(* PLC project Automating ships steam boiler, TK TC6_v0200_Example2 v2.0, author Toni Kucic *)
(* stored: creationDateTime 2019-09-29T20:50:27.2524554, version 4.1, modificationDateTime 2019-09-29T20:50:02.7007048, organization TkAutomation *)
(* Visit: https://github.com/tkucic/AutoSteamBoiler for more information. *)

TYPE BistableControlAPI_In_Typ : STRUCT
  DeactivateCmd : BOOL;  (* Deactivate cmd *)
  ActivateCmd : BOOL;  (* Activate cmd *)
END_STRUCT;
END_TYPE

TYPE BistableControlAPI_Out_Typ : STRUCT
  Deactivated : BOOL;  (* Device is deactivated *)
  Activated : BOOL;  (* Device is activated *)
  PositionError : BOOL;  (* TRUE: Object has position error *)
  Status : ARRAY[1..20] OF DINT;  (* 1:Open/Closed/InTransit, 2:OpenFail, 3:CloseFail, 4:FBError, 5:Control Position, 6:OpenCmd, 7:CloseCmd *)
  Icon : STRING;
END_STRUCT;
END_TYPE

TYPE BistableControlHMI_In_Typ : STRUCT
  DeactivateCmd : BOOL;  (* Deactivate cmd *)
  ActivateCmd : BOOL;  (* Activate cmd *)
  SetToAuto : BOOL;  (* Sets control to logic mode *)
  SetToMan : BOOL;  (* Sets control to HMI mode *)
END_STRUCT;
END_TYPE

TYPE BistableControlInit_Typ : STRUCT
  OpenFailDelay : TIME := TIME#6s0ms;  (* Open fail delay *)
  CloseFailDelay : TIME := TIME#6s0ms;  (* Close fail delay *)
  PositionErrorDelay : TIME := TIME#10s0ms;  (* Position error delay *)
  FBs : DWORD := 16#3;  (* B0 - Opened signal in use, B1 - Closed signal in use *)
END_STRUCT;
END_TYPE

TYPE BistableControlIO_In_Typ : STRUCT
  Deactivated : BOOL;  (* IO Open signal feedback from the device *)
  Activated : BOOL;  (* IO Close signal feedback from the device *)
  Tripped : BOOL;
  ReadyToOperate : BOOL := TRUE;
  Remote : BOOL := TRUE;
END_STRUCT;
END_TYPE

TYPE BistableControlIO_Out_Typ : STRUCT
  DeactivateCmd : BOOL;  (* IO deactivate command signal *)
  ActivateCmd : BOOL;  (* IO activate command signal *)
END_STRUCT;
END_TYPE

TYPE BistableIndAPI_Typ : STRUCT
  Deactivated : BOOL;  (* Device is deactivated *)
  Activated : BOOL;  (* Device is activated *)
  PositionError : BOOL;  (* TRUE: Object has position error *)
  Icon : STRING;
END_STRUCT;
END_TYPE

TYPE BistableIndInit_Typ : STRUCT
  PositionErrorDelay : TIME := TIME#10s0ms;  (* Position error alarm delay *)
  FBs : DWORD := 3;  (* B0 - Opened signal in use, B1 - Closed signal in use *)
END_STRUCT;
END_TYPE

TYPE BistableIndIO_In_Typ : STRUCT
  Deactivated : BOOL;  (* Device is deactivated input *)
  Activated : BOOL;  (* Device is activated input *)
  Tripped : BOOL;
END_STRUCT;
END_TYPE

TYPE DutyStandbyClassAPI_IN_Typ : STRUCT

END_STRUCT;
END_TYPE

TYPE DutyStandbyClassAPI_OUT_Typ : STRUCT

END_STRUCT;
END_TYPE

TYPE DutyStandbyClassInit_Typ : STRUCT

END_STRUCT;
END_TYPE

TYPE DutyStandbyClassIO_IN_Typ : STRUCT
  Pump1 : BistableControlIO_In_Typ;
  Pump2 : BistableControlIO_In_Typ;
END_STRUCT;
END_TYPE

TYPE DutyStandbyClassIO_OUT_Typ : STRUCT
  Pump1 : BistableControlIO_Out_Typ;
  Pump2 : BistableControlIO_Out_Typ;
END_STRUCT;
END_TYPE

TYPE TankControlClassAPI_IN_Typ : STRUCT
  LevelRef_pc : REAL;
END_STRUCT;
END_TYPE

TYPE TankControlClassAPI_OUT_Typ : STRUCT
  TankLevel_pc : REAL;
END_STRUCT;
END_TYPE

TYPE TankControlClassInit_Typ : STRUCT
  DrainValve : BistableControlInit_Typ;
  FillingValve : BistableControlInit_Typ;
END_STRUCT;
END_TYPE

TYPE TankControlClassIO_IN_Typ : STRUCT
  DrainValve : BistableControlIO_In_Typ;
  FillingValve : BistableControlIO_In_Typ;
  HLimitSwitch : BOOL;
  LLimitSwitch : BOOL;
  Level_cbm : REAL;
END_STRUCT;
END_TYPE

TYPE TankControlClassIO_OUT_Typ : STRUCT
  DrainValve : BistableControlIO_Out_Typ;
  FillingValve : BistableControlIO_Out_Typ;
END_STRUCT;
END_TYPE

TYPE AI_CFG_Typ : STRUCT
  sigMin : REAL;  (* Minimum value of the signal for scaling integer to real *)
  sigMax : REAL;  (* Maximum value of the signal for scaling integer to real *)
  Scale : REAL;  (* Scaling value of the signal for scaling integer to real *)
END_STRUCT;
END_TYPE

TYPE AI_IO_Typ : STRUCT
  PV_IN : REAL;  (* Input variable *)
  Status : DWORD;  (* Signal status *)
  AlarmHigh : BOOL;  (* High alarm flag *)
  AlarmHighHigh : BOOL;  (* High High alarm flag *)
  AlarmLow : BOOL;  (* Low alarm flag *)
  AlarmLowLow : BOOL;  (* Low Low alarm flag *)
  PV : REAL;  (* Proces variable *)
END_STRUCT;
END_TYPE

TYPE AO_CFG_Typ : STRUCT
  sigMin : REAL;  (* Minimum value of the signal for scaling integer to real *)
  sigMax : REAL;  (* Maximum value of the signal for scaling integer to real *)
  Scale : REAL;  (* Scaling value of the signal for scaling integer to real *)
END_STRUCT;
END_TYPE

TYPE AO_IO_Typ : STRUCT
  PV_IN : REAL;  (* Input variable *)
  Status : DWORD;  (* Signal status *)
  PV : REAL;  (* Proces variable *)
END_STRUCT;
END_TYPE

TYPE DI_CFG_Typ : STRUCT
  dummy1 : BOOL;
  dummy2 : BOOL;
  dummy3 : BOOL;
END_STRUCT;
END_TYPE

TYPE DI_IO_Typ : STRUCT
  Status : DWORD;  (* Signal status *)
  AlarmHigh : BOOL;  (* High alarm flag *)
  AlarmHighHigh : BOOL;  (* High High alarm flag *)
  AlarmLow : BOOL;  (* Low alarm flag *)
  AlarmLowLow : BOOL;  (* Low Low alarm flag *)
  PV : BOOL;  (* Proces variable *)
END_STRUCT;
END_TYPE

TYPE DO_CFG_Typ : STRUCT
  dummy1 : BOOL;
  dummy2 : BOOL;
  dummy3 : BOOL;
END_STRUCT;
END_TYPE

TYPE DO_IO_Typ : STRUCT
  Status : DWORD;  (* Signal status *)
  PV : BOOL;  (* Proces variable *)
END_STRUCT;
END_TYPE

TYPE IO_Typ : STRUCT
  AIS : AIS_Typ;  (* Analog input structure *)
  AOS : AOS_Typ;  (* Analog output structure *)
  DIS : DIS_Typ;  (* Digital input structure *)
  DOS : DOS_Typ;  (* Digital output structure *)
END_STRUCT;
END_TYPE

TYPE LIO : STRUCT
  IgnitionSeq : INT;
  ResetRequired : BOOL;
  FlameEstablished : BOOL;
  SteamCondensation : REAL;
  MasterFWPP : DINT;
  SteamDump : REAL;
  SteamConsumers : REAL;
END_STRUCT;
END_TYPE

TYPE AIS_Typ : STRUCT
  x150_BOILER_WATER_LEVEL : AI_IO_Typ;  (* Boiler water level *)
  x200_FRESH_WATER_STORAGE_TANK_LEVEL : AI_IO_Typ;  (* Fresh water storage tank level *)
  x200_FRESH_WATER_SERVICE_TANK_LEVEL : AI_IO_Typ;  (* Fresh water service tank level *)
  x300_HFO_HEATING_SYSTEM_CONSUMPTION : AI_IO_Typ;  (* HFO Heating system consumption *)
  x300_HVAC_SYSTEM_CONSUMPTION : AI_IO_Typ;  (* HVAC system consumption *)
  x300_OPERATIONAL_CONSUMERS_CONSUMPTION : AI_IO_Typ;  (* Operational consumers consumption *)
  x300_SYSTEM_STEAM_PRESSURE : AI_IO_Typ;  (* System steam pressure *)
END_STRUCT;
END_TYPE

TYPE AOS_Typ : STRUCT
  x150_BOILER_WATER_FEED_REGULATION_VALVE_SETPOINT : AO_IO_Typ;  (* Boiler water feed regulation valve setpoint *)
  x150_STEAM_DUMP_VALVE_SETPOINT : AO_IO_Typ;  (* Steam dump valve setpoint *)
  x100_AIR_VALVE_SETPOINT : AO_IO_Typ;  (* Air valve setpoint *)
  x100_FUEL_VALVE_SETPOINT : AO_IO_Typ;  (* Fuel valve setpoint *)
END_STRUCT;
END_TYPE

TYPE DOS_Typ : STRUCT
  x200_FW_SERVICE_PUMP1_STARTCMD : DO_IO_Typ;  (* Fresh water service pump 1 start command *)
  x200_FW_SERVICE_PUMP1_STOPCMD : DO_IO_Typ;  (* Fresh water service pump 1 stop command *)
  x200_FW_SERVICE_PUMP2_STARTCMD : DO_IO_Typ;  (* Fresh water service pump 2 start command *)
  x200_FW_SERVICE_PUMP2_STOPCMD : DO_IO_Typ;  (* Fresh water service pump 2 stop command *)
  x200_FW_STORAGE_TANK_DRAINVALVE_CLOSECMD : DO_IO_Typ;  (* Fresh water storage tank drain valve close command *)
  x200_FW_STORAGE_TANK_DRAINVALVE_OPENCMD : DO_IO_Typ;  (* Fresh water storage tank drain valve open command *)
  x200_FW_STORAGE_TANK_FILLVALVE_CLOSECMD : DO_IO_Typ;  (* Fresh water storage tank filling valve close command *)
  x200_FW_STORAGE_TANK_FILLVALVE_OPENCMD : DO_IO_Typ;  (* Fresh water storage tank filling valve open command *)
  x200_FW_SERVICE_TANK_DRAINVALVE_CLOSECMD : DO_IO_Typ;  (* Fresh water service tank drain valve close command *)
  x200_FW_SERVICE_TANK_DRAINVALVE_OPENCMD : DO_IO_Typ;  (* Fresh water service tank drain valve open command *)
  x200_FW_SERVICE_TANK_FILLVALVE_CLOSECMD : DO_IO_Typ;  (* Fresh water service tank filling valve close command *)
  x200_FW_SERVICE_TANK_FILLVALVE_OPENCMD : DO_IO_Typ;  (* Fresh water service tank filling valve open command *)
  x100_IGNITOR_ACTIVATE_CMD : DO_IO_Typ;  (* Ignitor activate cmd *)
  x100_BLOWER_MOTOR_START_CMD : DO_IO_Typ;  (* Blower motor start cmd *)
  x100_MAIN_FUEL_VALVE_CLOSE_CMD : DO_IO_Typ;  (* Main fuel valve close cmd *)
  x100_MAIN_FUEL_VALVE_OPEN_CMD : DO_IO_Typ;  (* Main fuel valve open cmd *)
  x300_HFO_HEATING_VALVE_CLOSE_CMD : DO_IO_Typ;  (* HFO heating valve close cmd *)
  x300_HFO_HEATING_VALVE_OPEN_CMD : DO_IO_Typ;  (* HFO heating valve open cmd *)
  x300_HVAC_HEATING_VALVE_CLOSE_CMD : DO_IO_Typ;  (* HVAC heating valve close cmd *)
  x300_HVAC_HEATING_VALVE_OPEN_CMD : DO_IO_Typ;  (* HVAC heating valve open cmd *)
  x300_OPERATIONAL_CONSUMERS_VALVE_CLOSE_CMD : DO_IO_Typ;  (* Operational consumers valve close cmd *)
  x300_OPERATIONAL_CONSUMERS_VALVE_OPEN_CMD : DO_IO_Typ;  (* Operational consumers valve open cmd *)
END_STRUCT;
END_TYPE

TYPE DIS_Typ : STRUCT
  x100_PHOTOCELL1_ACTIVE : DI_IO_Typ;  (* Photocell1Active *)
  x100_PHOTOCELL2_ACTIVE : DI_IO_Typ;  (* Photocell2Active *)
  x100_BURNER_DOOR_OPEN : DI_IO_Typ;  (* Burner door open *)
  x100_IGNITION_COIL_ACTIVATED : DI_IO_Typ;  (* Ignition coil activated *)
  x100_MAIN_FUEL_VALVE_CLOSED : DI_IO_Typ;  (* Main fuel valve closed *)
  x100_MAIN_FUEL_VALVE_OPEN : DI_IO_Typ;  (* Main fuel valve open *)
  x200_FW_STORAGE_TK_HLIMITSWITCH : DI_IO_Typ;  (* Fresh water storage tank high limit switch active *)
  x200_FW_STORAGE_TK_LLIMITSWITCH : DI_IO_Typ;  (* Fresh water storage tank low limit switch active *)
  x200_FW_SERVICE_PUMP2_RUNNING : DI_IO_Typ;  (* Fresh water service pump 2 running *)
  x200_FW_SERVICE_PUMP2_STOPPED : DI_IO_Typ;  (* Fresh water service pump 2 stopped *)
  x200_FW_SERVICE_PUMP2_READY : DI_IO_Typ;  (* Fresh water service pump 2 ready *)
  x200_FW_SERVICE_PUMP2_TRIPPED : DI_IO_Typ;  (* Fresh water service pump 2 tripped *)
  x200_FW_SERVICE_PUMP2_REMOTE : DI_IO_Typ;  (* Fresh water service pump 2 remote *)
  x200_FW_SERVICE_PUMP1_RUNNING : DI_IO_Typ;  (* Fresh water service pump 1 running *)
  x200_FW_SERVICE_PUMP1_STOPPED : DI_IO_Typ;  (* Fresh water service pump 1 stopped *)
  x200_FW_SERVICE_PUMP1_READY : DI_IO_Typ;  (* Fresh water service pump 1 ready *)
  x200_FW_SERVICE_PUMP1_TRIPPED : DI_IO_Typ;  (* Fresh water service pump 1 tripped *)
  x200_FW_SERVICE_PUMP1_REMOTE : DI_IO_Typ;  (* Fresh water service pump 1 remote *)
  x200_FW_STORAGE_TK_DRAINVALVE_CLOSED : DI_IO_Typ;  (* Fresh water storage tank drain valve closed *)
  x200_FW_STORAGE_TK_DRAINVALVE_OPENED : DI_IO_Typ;  (* Fresh water storage tank drain valve opened *)
  x200_FW_STORAGE_TK_DRAINVALVE_READY : DI_IO_Typ;  (* Fresh water storage tank drain valve ready *)
  x200_FW_STORAGE_TK_DRAINVALVE_REMOTE : DI_IO_Typ;  (* Fresh water storage tank drain valve remote *)
  x200_FW_STORAGE_TK_FILLVALVE_CLOSED : DI_IO_Typ;  (* Fresh water storage tank filling valve closed *)
  x200_FW_STORAGE_TK_FILLVALVE_OPENED : DI_IO_Typ;  (* Fresh water storage tank filling valve opened *)
  x200_FW_STORAGE_TK_FILLVALVE_READY : DI_IO_Typ;  (* Fresh water storage tank filling valve ready *)
  x200_FW_STORAGE_TK_FILLVALVE_REMOTE : DI_IO_Typ;  (* Fresh water storage tank filling valve remote *)
  x200_FW_SERVICE_TK_HLIMITSWITCH : DI_IO_Typ;  (* Fresh water service tank high limit switch active *)
  x200_FW_SERVICE_TK_LLIMITSWITCH : DI_IO_Typ;  (* Fresh water service tank low limit switch active *)
  x200_FW_SERVICE_TK_DRAINVALVE_CLOSED : DI_IO_Typ;  (* Fresh water service tank drain valve closed *)
  x200_FW_SERVICE_TK_DRAINVALVE_OPENED : DI_IO_Typ;  (* Fresh water service tank drain valve opened *)
  x200_FW_SERVICE_TK_DRAINVALVE_READY : DI_IO_Typ;  (* Fresh water service tank drain valve ready *)
  x200_FW_SERVICE_TK_DRAINVALVE_REMOTE : DI_IO_Typ;  (* Fresh water service tank drain valve remote *)
  x200_FW_SERVICE_TK_FILLVALVE_CLOSED : DI_IO_Typ;  (* Fresh water service tank filling valve closed *)
  x200_FW_SERVICE_TK_FILLVALVE_OPENED : DI_IO_Typ;  (* Fresh water service tank filling valve opened *)
  x200_FW_SERVICE_TK_FILLVALVE_READY : DI_IO_Typ;  (* Fresh water service tank filling valve ready *)
  x200_FW_SERVICE_TK_FILLVALVE_REMOTE : DI_IO_Typ;  (* Fresh water service tank filling valve remote *)
  x300_OPERATIONAL_CONSUMERS_VALVE_OPEN : DI_IO_Typ;  (* Operational consumers valve open *)
  x300_HFO_HEATING_VALVE_CLOSED : DI_IO_Typ;  (* HFO heating valve closed *)
  x300_HFO_HEATING_VALVE_OPEN : DI_IO_Typ;  (* HFO heating valve open *)
  x300_HVAC_HEATING_VALVE_CLOSED : DI_IO_Typ;  (* HVAC heating valve closed *)
  x300_HVAC_HEATING_VALVE_OPEN : DI_IO_Typ;  (* HVAC heating valve open *)
  x300_OPERATIONAL_CONSUMERS_VALVE_CLOSED : DI_IO_Typ;  (* Operational consumers valve closed *)
  x900_EMERGENCY_STOP : DI_IO_Typ;  (* Emergency stop *)
  x900_SYSTEM_REMOTE_SWITCH : DI_IO_Typ;  (* SystemRemote switch *)
END_STRUCT;
END_TYPE

TYPE SimCFG : STRUCT
  BlinkFreq : TIME := TIME#500ms;
  FWTankLSHighTrig : REAL := 85;
  FWTankLSHighHighTrig : REAL := 95;
  FWTankLSLowTrig : REAL := 15;
  FWTankLSLowLowTrig : REAL := 5;
  SteamFactor : REAL := 0.021;
  ReliefValveOpeningSP : REAL := 35;
  Inflow : REAL := 0.11;
  WaterEvapFactor : REAL := 0.06;
  MaxDump : REAL := 1;
  OverpressureMultiplier : REAL := 1;
  DrainTankMultiplier : REAL := 0.5;
  PCell1DetectDelay : TIME := TIME#500ms;
  PCell2DetectDelay : TIME := TIME#1s0ms;
  ValveOperatingTime : TIME := TIME#3s0ms;
  LostWaterOnConsumers : REAL := 0.1;
END_STRUCT;
END_TYPE

TYPE CFG_Typ : STRUCT
  FWTankHighLimit : REAL := 90;  (* High water level limit *)
  FWTankLowLimit : REAL := 30;  (* Low water level limit *)
  FWTankLowTrip : REAL := 15;
  FWTankLowAlarmDelay : TIME := TIME#1s0ms;
  SteamPressureSP : REAL := 7;  (* Setpoint for system steam pressure *)
  FWServiceTKSP : REAL := 70;  (* Setpoint for the FW Service tank water level *)
  SteamPressHighTrip : REAL := 45;
  SteamPressHighLimit : REAL := 8.5;  (* High steam pressure limit *)
  SteamPressLowLimit : REAL := 1;  (* Low steam pressure limit *)
  SteamPressHighAlarmDelay : TIME := TIME#1s0ms;
  FuelValveStart_pc : REAL := 10;  (* Starting valve opening upon ignition sequence *)
  DualPumpsTimer : TIME := TIME#5s0ms;  (* Time for FW pumps to run in paralel during sw/o *)
  BlowingOutTime : TIME := TIME#10s0ms;  (* Time for safety blow out of burner *)
  IgnitionFailDelay : TIME := TIME#5s0ms;  (* Time before ignition fail occurs *)
  MainFuelValveOperationDelay : TIME := TIME#5s0ms;
  F_PID_P : REAL := 1.5;
  F_PID_I : REAL := 0.9;
  F_PID_D : REAL := 0;
  F_PID_Offset : REAL := 0;
  F_PID_OutMIN : REAL := 2.1;
  F_PID_OutMAX : REAL := 100;
  AirToFuelRatio : REAL := 1.25;
  W_PID_P : REAL := 1.5;
  W_PID_I : REAL := 0.9;
  W_PID_D : REAL := 0;
  W_PID_Offset : REAL := 0;
  HFOConsumerNominal : REAL := 1;
  HFOHeatValveOperDelay : TIME := TIME#5s0ms;
  HVACConsumerNominal : REAL := 0.5;
  HVACHeatValveOperDelay : TIME := TIME#5s0ms;
  OperConsumerNominal : REAL := 0.65;
  OperConsValveOperDelay : TIME := TIME#5s0ms;
  S_PID_P : REAL := -1.5;
  S_PID_I : REAL := 0.9;
  S_PID_D : REAL := 0;
  TxtRemote : STRING := 'REMOTE';
  TxtManual : STRING := 'MANUAL';
  TxtOvrFl : STRING := 'FW Tank overflowing';
  TxtFWTkEmpty : STRING := 'FW Tank empty';
  TxtSysReady : STRING := 'System ready for operation';
  TxtSysBlow : STRING := 'System blowout begun';
  TxtIgnite : STRING := 'Igniting burner';
  TxtSysRun : STRING := 'System running';
  TxtIgnFail : STRING := 'Ignition failed';
  TxtEmcyStp : STRING := 'Emergency stop active';
  TxtAbort : STRING := 'Operation aborted by user';
  TxtSysNotReady : STRING := 'System not ready';
END_STRUCT;
END_TYPE

TYPE Vars : STRUCT
  CFG : CFG_Typ;
  dummy1 : BOOL;
  dummy2 : BOOL;
END_STRUCT;
END_TYPE

FUNCTION_BLOCK BurnerControlClass

            
          
END_FUNCTION_BLOCK

FUNCTION_BLOCK fbAuxDevCtrl
  VAR
    ChangeOverTrig : R_TRIG;
    DualPumpsTimer : TOn;
    WaterLevelCTRL : PID;
    vManual : REAL;
    vPIDOFF : BOOL;
    vReset : BOOL;
    vLimitsActive : BOOL;
    vPIDOverflow : BOOL;
  END_VAR
  VAR RETAIN
    vMasterFWPP : INT := 1;
    vAutoStopFWPump2 : BOOL;
    vAutoStartFWPump2 : BOOL;
    vAutoStopFWPump1 : BOOL;
    vAutoStartFWPump1 : BOOL;
    vFWTkSP : REAL := 75;
  END_VAR

            // (* Switch Water level PID off if tank is overflowing *)
// vPIDOFF := GVL.IO.DIS.FWTankLSHighHigh OR GVL.IO.AIS.FWTank_Level > GVL.CFG_Typ.FWTankHighLimit;
// 
// (* Change over functionality. This switches the pumps.*)
// ChangeOverTrig(CLK:=GVL.IO.DIS.FWChangeOverPP);
// 
// IF vMasterFWPP = 1 AND ChangeOverTrig.Q THEN
// 	vMasterFWPP := 2;
// ELSIF vMasterFWPP = 2 AND ChangeOverTrig.Q THEN
// 	vMasterFWPP := 1;
// END_IF;
// 
// (* Automatic regulation of fresh water service tanks level *)
// IF GVL.IO.DIS.RemoteFWPP THEN
// 	vAutoStopFWPump1 := (vMasterFWPP = 1) AND (GVL.IO.DIS.FWTankLSHigh OR GVL.IO.DIS.FWTankLSHighHigh) AND GVL.IO.DOS_Typ.FWPump1;
// 	vAutoStartFWPump1 := (vMasterFWPP = 1) AND (GVL.IO.DIS.FWTankLSLow OR GVL.IO.DIS.FWTankLSLowLow) AND NOT GVL.IO.DOS_Typ.FWPump1;
// 	vAutoStopFWPump2 := (vMasterFWPP = 2) AND (GVL.IO.DIS.FWTankLSHigh OR GVL.IO.DIS.FWTankLSHighHigh) AND GVL.IO.DOS_Typ.FWPump2;
// 	vAutoStartFWPump2 := (vMasterFWPP = 2) AND (GVL.IO.DIS.FWTankLSLow OR GVL.IO.DIS.FWTankLSLowLow) AND NOT GVL.IO.DOS_Typ.FWPump2;
// ELSE
// 	vAutoStopFWPump1 := (vMasterFWPP = 1) AND (GVL.IO.DIS.FWManStop OR GVL.IO.DIS.FWTankLSHighHigh) AND GVL.IO.DOS_Typ.FWPump1;
// 	vAutoStartFWPump1 := (vMasterFWPP = 1) AND GVL.IO.DIS.FWManStart AND NOT GVL.IO.DOS_Typ.FWPump1;
// 	vAutoStopFWPump2 := (vMasterFWPP = 2) AND (GVL.IO.DIS.FWManStop OR GVL.IO.DIS.FWTankLSHighHigh) AND GVL.IO.DOS_Typ.FWPump2;
// 	vAutoStartFWPump2 := (vMasterFWPP = 2) AND GVL.IO.DIS.FWManStart AND NOT GVL.IO.DOS_Typ.FWPump2;
// END_IF
// 
// (*Pumps run paralel for some time to not lose pressure *)
// IF vMasterFWPP = 2 AND GVL.IO.DIS.FWServicePump1=1 THEN
// 	GVL.IO.DOS_Typ.FWPump2 := TRUE;
// 
// 	DualPumpsTimer(IN:=TRUE, PT:=GVL.CFG_Typ.DualPumpsTimer);
// 	IF DualPumpsTimer.Q THEN
// 		GVL.IO.DOS_Typ.FWPump1 := FALSE;
// 		DualPumpsTimer(IN:=FALSE);
// 	END_IF
// ELSIF vAutoStartFWPump1 THEN
// 	GVL.IO.DOS_Typ.FWPump1 := TRUE;
// ELSIF vAutoStopFWPump1 THEN
// 	GVL.IO.DOS_Typ.FWPump1 := FALSE;
// END_IF
// 
// IF vMasterFWPP = 1 AND GVL.IO.DIS.FWServicePump2=1 THEN
// 	GVL.IO.DOS_Typ.FWPump1 := TRUE;
// 	
// 	DualPumpsTimer(IN:=TRUE, PT:=GVL.CFG_Typ.DualPumpsTimer);
// 	IF DualPumpsTimer.Q THEN
// 		GVL.IO.DOS_Typ.FWPump2 := FALSE;
// 		DualPumpsTimer(IN:=FALSE);
// 	END_IF
// ELSIF vAutoStartFWPump2 THEN
// 	GVL.IO.DOS_Typ.FWPump2 := TRUE;
// ELSIF vAutoStopFWPump2 THEN
// 	GVL.IO.DOS_Typ.FWPump2 := FALSE;
// END_IF
// 
// WaterLevelCTRL(
// 	ACTUAL:= GVL.IO.AIS.FWTank_Level, 
// 	SET_POINT:= GVL.CFG_Typ.FWServiceTKSP, 
// 	KP:= GVL.CFG_Typ.W_PID_P, 
// 	TN:= GVL.CFG_Typ.W_PID_I, 
// 	TV:= GVL.CFG_Typ.W_PID_D, 
// 	Y_MANUAL:= 0, 
// 	Y_OFFSET:= GVL.CFG_Typ.W_PID_Offset, 
// 	Y_MIN:= 0, 
// 	Y_MAX:= 100, 
// 	MANUAL:= vPIDOFF, 
// 	RESET:= vReset, 
// 	Y=> GVL.IO.AOS.FWTkRegValve, 
// 	LIMITS_ACTIVE=> vLimitsActive, 
// 	OVERFLOW=> vPIDOverflow);
// 
// (* Send system status to other programs *)
// GVL.LIO.MasterFWPP := vMasterFWPP;
          
END_FUNCTION_BLOCK

FUNCTION_BLOCK fbBoilerSystem

            
          
END_FUNCTION_BLOCK

FUNCTION_BLOCK fbStateMachine
  VAR
    BlowingTimeTimer : TON;
    DelayTimer : TON;
    AutoStartSR : SR;
    vFlameOut : BOOL;
    vOpenMainFuelValveCmd : BOOL;  (* MainFuelValveCtrl: OnOffValve_Object; *)
    vCloseMainFuelValveCmd : BOOL;
    vCloseMainFuelValveHMI : BOOL;
    vOpenMainFuelValveHMI : BOOL;
    vSetMainFuelValveToAuto : BOOL;
    vSetMainFuelValveToMan : BOOL;
    vMainFuelValveStatus : ARRAY[1..20] OF DINT;
    vMainFuelValveIcon : STRING;
    vMainFuelValveButton : BOOL;
  END_VAR
  VAR CONSTANT
    cStateNotReady : INT := 0;
    cStateStandby : INT := 1;
    cStateAirBlowing : INT := 2;
    cStateIgnition : INT := 3;
    cStateSystemIgnited : INT := 4;
    cStateIgnitionFail : INT := 10;
    cStateEmergencyStop : INT := 11;
    cStateUserAbort : INT := 12;
  END_VAR
  VAR RETAIN
    vSequence : INT := 0;
    vSequenceDone : INT;
    vIgnTimerStart : BOOL;
    vIgnSeqStart : BOOL;
    vMessage : STRING(INT#50);
    vResetRequired : BOOL;
    vAutoStart : BOOL;
    vFWTankLowTrip : BOOL;
    vHighPressureTrip : BOOL;
  END_VAR

            // (*******************************************)
// (* 0 - System not ready                    *)
// (* 1 - System standby                      *)
// (* 2 - Air blowing                         *)
// (* 3 - Ignition                            *)
// (* 4 - System ignited                      *)
// (* 10 - Ignition fail                      *)
// (* 11 - Emergency stop                     *)
// (* 12 - User abort                         *)
// (*******************************************)
// 
// (* Safety tripping *)
// 
// vFWTankLowTrip := GVL.IO.AIS.FWTank_Level < GVL.CFG_Typ.FWTankLowTrip AND (vSequence = cStateSystemIgnited);
// 
// vHighPressureTrip := GVL.IO.AIS.SteamPressure > GVL.CFG_Typ.SteamPressHighLimit;
// 
// vFlameOut := (vSequence = cStateSystemIgnited) AND NOT (GVL.IO.DIS.Photocell1 OR GVL.IO.DIS.Photocell2);
// 
// IF vFWTankLowTrip OR vHighPressureTrip OR vFlameOut OR GVL.IO.DIS.BurnerOpen THEN
// 	vSequence := cStateEmergencyStop;
// END_IF
// 
// IF  NOT GVL.IO.DIS.EmcyStopPB THEN
// 	vSequence := cStateEmergencyStop;
// END_IF
// 
// AutoStartSR(Set1:= (GVL.IO.AIS.SteamPressure < GVL.CFG_Typ.SteamPressureSP AND vSequence = cStateStandby), 
// 			Reset:= vSequence <> cStateStandby,
// 			Q1 => vAutoStart);
// 
// CASE vSequence OF
// 		10,11,12: vResetRequired := TRUE;
// ELSE
// 		vResetRequired := FALSE;
// END_CASE
// 
// CASE vSequence OF
// 	
// 	(* System not ready *)
// 	0: vMessage := GVL.CFG_Typ.TxtSysNotReady;
// 		IF GVL.IO.AIS.FWTank_Level > GVL.CFG_Typ.FWTankLowLimit AND GVL.IO.AIS.SteamPressure < GVL.CFG_Typ.SteamPressHighLimit THEN
// 			vSequence := cStateStandby;
// 		END_IF
// 		vSequenceDone := 0;
// 
// 	(* System standby *)
// 	1:  vMessage := GVL.CFG_Typ.TxtSysReady;
// 		IF vAutoStart AND GVL.IO.DIS.RemoteSW THEN
// 			vSequence := cStateAirBlowing;
// 		ELSIF GVL.IO.DIS.ManStartPB THEN
// 			vSequence := cStateAirBlowing;
// 		END_IF
// 		vSequenceDone := 1;
// 		
// 	(* Air blowing and opening valves *)	
// 	2:  vMessage := GVL.CFG_Typ.TxtSysBlow;		
// 		BlowingTimeTimer(IN:=vSequenceDone = 2, PT := GVL.CFG_Typ.BlowingOutTime);
// 		
// 		vOpenMainFuelValveCmd := NOT GVL.IO.DIS.MainFuelValveOpen AND GVL.IO.DIS.RemoteSW;
// 		vCloseMainFuelValveCmd := FALSE;
// 		
// 		GVL.IO.DOS_Typ.AirBlowerMotor := TRUE;
// 		
// 		IF GVL.IO.DIS.StopPB THEN
// 			vSequence := cStateUserAbort;
// 		END_IF;	
// 		
// 		IF BlowingTimeTimer.Q AND GVL.IO.DIS.MainFuelValveOpen THEN
// 			vSequence := cStateIgnition;
// 		ELSIF BlowingTimeTimer.Q AND NOT GVL.IO.DIS.MainFuelValveOpen THEN
// 			vSequence := cStateIgnitionFail;
// 		END_IF
// 		vSequenceDone := 2;
// 	
// 	(* Ignition *)
// 	3:  vMessage := GVL.CFG_Typ.TxtIgnite;
// 		IF GVL.IO.DIS.StopPB THEN
// 			vSequence := cStateUserAbort;
// 		END_IF;	
// 	    vIgnSeqStart :=  vIgnSeqStart OR (GVL.IO.DIS.RemoteSW) OR (GVL.IO.DIS.ManIgnite);
// 		vIgnTimerStart := vSequenceDone = 3 AND vIgnSeqStart;
// 
// 		DelayTimer(IN := vIgnTimerStart, PT := GVL.CFG_Typ.IgnitionFailDelay);
// 		IF DelayTimer.Q THEN
// 			vSequence := cStateIgnitionFail;
// 		END_IF
// 		IF vIgnSeqStart THEN
// 			GVL.IO.DOS_Typ.Ignitor := TRUE;
// 			IF GVL.IO.DIS.Photocell1 OR GVL.IO.DIS.Photocell2 THEN
// 				vSequence := cStateSystemIgnited;
// 				GVL.IO.DIS.ManIgnite := FALSE;
// 				GVL.IO.DOS_Typ.Ignitor := FALSE;
// 				vIgnSeqStart := FALSE;
// 			END_IF
// 		END_IF;
// 		vSequenceDone := 3;
// 		
// 	(* System ignited *)	
// 	4:	vMessage := GVL.CFG_Typ.TxtSysRun;
// 		IF GVL.IO.DIS.StopPB THEN
// 			vSequence := cStateUserAbort;
// 		END_IF;	
// 		vSequenceDone := 4;
// 		
// 	(* Ignition fail *)	
// 	10: vMessage := GVL.CFG_Typ.TxtIgnFail;
// 		GVL.IO.DOS_Typ.Ignitor := FALSE;		
// 		vOpenMainFuelValveCmd := FALSE;
// 		vCloseMainFuelValveCmd := TRUE;
// 		IF GVL.IO.DIS.Reset THEN
// 			vSequence := cStateNotReady;
// 		END_IF
// 		vSequenceDone := 10;
// 		
// 	(* Emergency stop *)	
// 	11: vMessage := GVL.CFG_Typ.TxtEmcyStp;
// 		GVL.IO.DOS_Typ.Ignitor := FALSE;		
// 		vOpenMainFuelValveCmd := FALSE;
// 		vCloseMainFuelValveCmd := TRUE;
// 		IF GVL.IO.DIS.Reset AND GVL.IO.DIS.EmcyStopPB THEN
// 			vSequence := cStateNotReady;
// 		END_IF	
// 		vSequenceDone := 11;
// 		
// 	(* User abort *)	
// 	12:	vMessage := GVL.CFG_Typ.TxtAbort;
// 		BlowingTimeTimer(IN := vSequenceDone = 12, PT := GVL.CFG_Typ.BlowingOutTime);
// 		IF NOT BlowingTimeTimer.Q THEN
// 			GVL.IO.DOS_Typ.AirBlowerMotor := TRUE;
// 		ELSE
// 			GVL.IO.DOS_Typ.AirBlowerMotor := FALSE;
// 		END_IF
// 		IF GVL.IO.DIS.Reset THEN
// 			vSequence := cStateNotReady;
// 		END_IF
// 		GVL.IO.DOS_Typ.Ignitor := FALSE;	
// 		vOpenMainFuelValveCmd := FALSE;
// 		vCloseMainFuelValveCmd := TRUE;
// 		vSequenceDone := 12;
// ELSE
// 	vSequence := cStateNotReady;
// END_CASE
// 
// IF vSequence <> 3 THEN
// 	GVL.IO.DIS.ManIgnite := FALSE;
// END_IF;
// 
// (* Send system status to other programs *)
// GVL.LIO.IgnitionSeq := vSequence;
// GVL.LIO.ResetRequired := vResetRequired;
// 
// (* Fuel Valve controllers *)
// 
// MainFuelValveCtrl(
// 	iOpenedFB:= GVL.IO.DIS.MainFuelValveOpen, 
// 	iClosedFB:= GVL.IO.DIS.MainFuelValveClosed, 
// 	OpenAutoCmd:= vOpenMainFuelValveCmd, 
// 	CloseAutoCmd:= vCloseMainFuelValveCmd, 
// 	OpenCmdHMI:= vOpenMainFuelValveHMI, 
// 	CloseCmdHMI:= vCloseMainFuelValveHMI, 
// 	SetToAuto:= vSetMainFuelValveToAuto, 
// 	SetToMan:= vSetMainFuelValveToMan, 
// 	cfgOpenFailDelay:= GVL.CFG_Typ.MainFuelValveOperationDelay, 
// 	cfgCloseFailDelay:= GVL.CFG_Typ.MainFuelValveOperationDelay, 
// 	cfgFBErrorDelay:= GVL.CFG_Typ.MainFuelValveOperationDelay, 
// 	ValveStatus=> vMainFuelValveStatus, 
// 	ValveIcon=> vMainFuelValveIcon, 
// 	qOpenCmd=> GVL.IO.DOS_Typ.FuelValveOpenCmd, 
// 	qCloseCmd=> GVL.IO.DOS_Typ.FuelValveCloseCmd);

          
END_FUNCTION_BLOCK

FUNCTION_BLOCK fbSteamControl
  VAR
    FuelController : PID;
    SteamDumpController : PID;
    rtManUp : R_TRIG;
    rtManDown : R_TRIG;
    vMan_Y : REAL;
    vHFOHeatOpenCmdHMI : BOOL;  (* HFOHeatValve: OnOffValve_Object; HVACHeatValve: OnOffValve_Object; OperConsValve: OnOffValve_Object; *)
    vHFOHeatCloseCmdHMI : BOOL;
    vHFOHeatSetToAuto : BOOL;
    vHFOHeatSetToMan : BOOL;
    vHFOHeatValveStatus : ARRAY[1..20] OF DINT;
    vHFOHeatValveIcon : STRING;
    vHFOHeatValveButton : BOOL;
    vHVACHeatOpenCmdHMI : BOOL;
    vHVACHeatCloseCmdHMI : BOOL;
    vHVACHeatSetToMan : BOOL;
    vHVACHeatValveStatus : ARRAY[1..20] OF DINT;
    vHVACHeatValveIcon : STRING;
    vHVACHeatValveButton : BOOL;
    vOperConsOpenCmdHMI : BOOL;
    vOperConsCloseCmdHMI : BOOL;
    vOperConsSetToMan : BOOL;
    vOperConsValveStatus : ARRAY[1..20] OF DINT;
    vOperConsValveIcon : STRING;
    vOperConsValveButton : BOOL;
    vHFOHeatOpenAutoCmd : BOOL;
    vHFOHeatCloseAutoCmd : BOOL;
    vHVACHeatValveOpenAutoCmd : BOOL;
    vHVACHeatValveCloseAutoCmd : BOOL;
    vHVACHeatSetToAuto : BOOL;
    vOperConsValveOpenAutoCmd : BOOL;
    vOperConsValveCloseAutoCmd : BOOL;
    vOperConsSetToAuto : BOOL;
  END_VAR
  VAR RETAIN
    vPIDManual : BOOL;
    vOverflow : BOOL;
    vPIDLimitActive : BOOL;
  END_VAR

            // IF GVL.LIO.IgnitionSeq > 4 OR GVL.LIO.IgnitionSeq = 0 THEN
// 	(* Switch off fuel valve *)
// 	vPIDManual	:= TRUE;
// 	vMan_Y		:= 0;
// 
// ELSIF GVL.LIO.IgnitionSeq = 3 THEN
// 	(* Stabilize ignition *)
// 	vPIDManual := TRUE;
// 	vMan_Y 	   := GVL.SysCFG.FuelValveStart_pc;
// 
// ELSIF GVL.LIO.IgnitionSeq = 4 THEN
// 	IF GVL.IO.DIS.RemoteSW THEN
// 		vPIDManual := FALSE;
// 		vMan_Y := GVL.IO.AOS.FuelValve;
// 	ELSIF NOT GVL.IO.DIS.RemoteSW THEN
// 		vPIDManual := TRUE;
// 		rtManUp(CLK:=GVL.IO.DIS.ManLoadUP);
// 		rtManDown(CLK:=GVL.IO.DIS.ManLoadDown);
// 	
// 		IF rtManUp.Q THEN
// 			vMan_Y := vMan_Y + 1;
// 		END_IF
// 		IF rtManDown.Q THEN
// 			vMan_Y := vMan_Y - 1;
// 		END_IF
// 	END_IF
// 		
// ELSE
// 	vPIDManual	:= TRUE;
// 	vMan_Y		:= 0;
// END_IF;
// 
// FuelController(
// 	ACTUAL:= GVL.IO.AIS.SteamPressure, 
// 	SET_POINT:= GVL.SysCFG.SteamPressureSP , 
// 	KP:= GVL.SysCFG.F_PID_P, 
// 	TN:= GVL.SysCFG.F_PID_I, 
// 	TV:= GVL.SysCFG.F_PID_D, 
// 	Y_MANUAL:= vMan_Y, 
// 	Y_OFFSET:= GVL.SysCFG.F_PID_Offset, 
// 	Y_MIN:= GVL.SysCFG.F_PID_OutMIN, 
// 	Y_MAX:= GVL.SysCFG.F_PID_OutMAX,
// 	MANUAL := vPIDManual,
// 	RESET:=FALSE , 
// 	Y=> GVL.IO.AOS.FuelValve, 
// 	LIMITS_ACTIVE=> vPIDLimitActive, 
// 	OVERFLOW=>vOverflow );
// 
// SteamDumpController(
// 	ACTUAL:= GVL.IO.AIS.SteamPressure, 
// 	SET_POINT:= GVL.SysCFG.SteamPressureSP , 
// 	KP:= GVL.SysCFG.S_PID_P, 
// 	TN:= GVL.SysCFG.S_PID_I, 
// 	TV:= GVL.SysCFG.S_PID_D, 
// 	Y_MIN:= 0, 
// 	Y_MAX:= 100,
// 	Y=> GVL.IO.AOS.SteamDumpValve);
// 	
// (* Consumer valve handling *)
// HFOHeatValve(
// 	iOpenedFB:= GVL.IO.DIS.HFOHeatValveOpen , 
// 	iClosedFB:= GVL.IO.DIS.HFOHeatValveClosed, 
// 	OpenAutoCmd:= vHFOHeatOpenAutoCmd, 
// 	CloseAutoCmd:= vHFOHeatCloseAutoCmd, 
// 	OpenCmdHMI:= vHFOHeatOpenCmdHMI, 
// 	CloseCmdHMI:= vHFOHeatCloseCmdHMI, 
// 	SetToAuto:= vHFOHeatSetToAuto, 
// 	SetToMan:= vHFOHeatSetToMan, 
// 	cfgOpenFailDelay:= GVL.SysCFG.HFOHeatValveOperDelay, 
// 	cfgCloseFailDelay:= GVL.SysCFG.HFOHeatValveOperDelay, 
// 	cfgFBErrorDelay:= GVL.SysCFG.HFOHeatValveOperDelay, 
// 	ValveStatus=> vHFOHeatValveStatus, 
// 	ValveIcon=> vHFOHeatValveIcon, 
// 	qOpenCmd=> GVL.IO.DOS.HFOHeatValveOpenCmd, 
// 	qCloseCmd=> GVL.IO.DOS.HFOHeatValveCloseCmd);
// 	
// HVACHeatValve(
// 	iOpenedFB:= GVL.IO.DIS.HVACHeatValveOpen , 
// 	iClosedFB:= GVL.IO.DIS.HVACHeatValveClosed, 
// 	OpenAutoCmd:= vHVACHeatValveOpenAutoCmd, 
// 	CloseAutoCmd:= vHVACHeatValveCloseAutoCmd, 
// 	OpenCmdHMI:= vHVACHeatOpenCmdHMI, 
// 	CloseCmdHMI:= vHVACHeatCloseCmdHMI, 
// 	SetToAuto:= vHVACHeatSetToAuto, 
// 	SetToMan:= vHVACHeatSetToMan, 
// 	cfgOpenFailDelay:= GVL.SysCFG.HVACHeatValveOperDelay, 
// 	cfgCloseFailDelay:= GVL.SysCFG.HVACHeatValveOperDelay, 
// 	cfgFBErrorDelay:= GVL.SysCFG.HVACHeatValveOperDelay, 
// 	ValveStatus=> vHVACHeatValveStatus, 
// 	ValveIcon=> vHVACHeatValveIcon, 
// 	qOpenCmd=> GVL.IO.DOS.HVACHeatValveOpenCmd, 
// 	qCloseCmd=> GVL.IO.DOS.HVACHeatValveCloseCmd);
// 	
// OperConsValve(
// 	iOpenedFB:= GVL.IO.DIS.OperConsValveOpen , 
// 	iClosedFB:= GVL.IO.DIS.OperConsValveClosed, 
// 	OpenAutoCmd:= vOperConsValveOpenAutoCmd, 
// 	CloseAutoCmd:= vOperConsValveCloseAutoCmd, 
// 	OpenCmdHMI:= vOperConsOpenCmdHMI, 
// 	CloseCmdHMI:= vOperConsCloseCmdHMI, 
// 	SetToAuto:= vOperConsSetToAuto, 
// 	SetToMan:= vOperConsSetToMan, 
// 	cfgOpenFailDelay:= GVL.SysCFG.OperConsValveOperDelay, 
// 	cfgCloseFailDelay:= GVL.SysCFG.OperConsValveOperDelay, 
// 	cfgFBErrorDelay:= GVL.SysCFG.OperConsValveOperDelay, 
// 	ValveStatus=> vOperConsValveStatus, 
// 	ValveIcon=> vOperConsValveIcon, 
// 	qOpenCmd=> GVL.IO.DOS.OperConsValveOpenCmd, 
// 	qCloseCmd=> GVL.IO.DOS.OperConsValveCloseCmd);
// 	
// (* Air flap opening *)
// GVL.IO.AOS.AirValve := GVL.IO.AOS.FuelValve / GVL.SysCFG.AirToFuelRatio;
// 

          
END_FUNCTION_BLOCK

FUNCTION_BLOCK BistableControlClass
  VAR_INPUT
    init : BistableControlInit_Typ;
    io_in : BistableControlIO_In_Typ;
    API_IN : BistableControlHMI_In_Typ;
    HMI_IN : BistableControlHMI_In_Typ;
  END_VAR
  VAR_OUTPUT
    HMI_OUT : BistableControlAPI_Out_Typ;
    API_OUT : BistableControlAPI_Out_Typ;
    io_out : BistableControlIO_Out_Typ;
  END_VAR
  VAR
    constructor : BistableIndicationClass;  (* Base building block of this object *)
    OpenFail : TON;
    CloseFail : TON;
    vControlPosition : DINT;
    vDeactivateCmd : BOOL;
    vActivateCmd : BOOL;
  END_VAR

            (* Handle base constructor *)
constructor.init.FBs := init.FBs;
constructor.init.PositionErrorDelay := init.PositionErrorDelay;
constructor.io_in.Activated := io_in.Activated;
constructor.io_in.Deactivated := io_in.Deactivated;
constructor.io_in.Tripped := io_in.Tripped;

constructor();

(* Control location *)
(* Auto/Man setting should be rtrig or non holding button *)
IF HMI_IN.SetToAuto AND NOT HMI_IN.SetToMan THEN
	vControlPosition := 1;
ELSIF HMI_IN.SetToMan THEN
	vControlPosition := 0;
END_IF

IF NOT(OpenFail.Q OR CloseFail.Q) THEN
	IF vControlPosition = 1 THEN
		vDeactivateCmd := (vDeactivateCmd OR HMI_IN.DeactivateCmd) AND NOT constructor.API.Deactivated;
		vActivateCmd := (vActivateCmd OR HMI_IN.ActivateCmd) AND NOT constructor.API.Activated;
	ELSIF vControlPosition = 0 THEN
		vDeactivateCmd := (vDeactivateCmd OR API_IN.DeactivateCmd) AND NOT constructor.API.Deactivated;
		vActivateCmd := (vActivateCmd OR API_IN.ActivateCmd) AND NOT constructor.API.Activated;
	ELSE
		vDeactivateCmd := FALSE;
		vActivateCmd := FALSE;	
	END_IF
ELSE
		vDeactivateCmd := FALSE;
		vActivateCmd := FALSE;		
END_IF

OpenFail(IN:= vDeactivateCmd AND NOT constructor.API.Deactivated, PT:= init.OpenFailDelay);
CloseFail(IN:= vActivateCmd AND NOT constructor.API.Activated, PT:= init.CloseFailDelay);

io_out.DeactivateCmd := vDeactivateCmd AND NOT (OpenFail.Q OR constructor.API.Deactivated OR constructor.API.PositionError);
io_out.ActivateCmd := vActivateCmd AND NOT (CloseFail.Q OR constructor.API.Activated OR constructor.API.PositionError);

API_OUT.Status[1] := BOOL_TO_DINT(constructor.API.Deactivated) + 2*BOOL_TO_DINT(constructor.API.Activated);
API_OUT.Status[2] := BOOL_TO_DINT(OpenFail.Q);
API_OUT.Status[3] := BOOL_TO_DINT(CloseFail.Q);
API_OUT.Status[4] := BOOL_TO_DINT(constructor.API.PositionError);
API_OUT.Status[5] := vControlPosition;
API_OUT.Status[6] := BOOL_TO_DINT(io_out.DeactivateCmd);
API_OUT.Status[7] := BOOL_TO_DINT(io_out.ActivateCmd);

IF API_OUT.Status[1] = 1 THEN
	API_OUT.Icon := 'Valve1';
ELSIF API_OUT.Status[1] = 2 THEN
	API_OUT.Icon := 'Valve2';
ELSE
	API_OUT.Icon := 'Valve3';
END_IF


          
END_FUNCTION_BLOCK

FUNCTION_BLOCK BistableIndicationClass
  VAR_INPUT
    init : BistableIndInit_Typ;  (* This classes initialization/config structure *)
    io_in : BistableIndIO_In_Typ;  (* This classes input signals *)
  END_VAR
  VAR_OUTPUT
    API : BistableIndAPI_Typ;  (* Communication structure to higher logic *)
    HMI : BistableIndAPI_Typ;  (* Communication structure to HMI *)
  END_VAR
  VAR
    PositionErrorDelay : TON;  (* Position error alarm delay *)
    vPositionErrorOld : BOOL;  (* Event memory: Position error *)
    vDeactivatedOld : BOOL;  (* Event memory: Deactivated *)
    vActivatedOld : BOOL;  (* Event memory: Activated *)
  END_VAR

            (* Handle IOs depending on init. *)
IF init.FBs.0 AND init.FBs.1 THEN
	API.Activated := io_in.Activated;
	API.Deactivated := io_in.Deactivated;
ELSIF init.FBs.0 THEN
	API.Activated := NOT io_in.Deactivated;
	API.Deactivated := io_in.Deactivated;
ELSIF init.FBs.1 THEN
	API.Activated := io_in.Activated;
	API.Deactivated := NOT io_in.Activated;
ELSE
	(* Invalid configuration *)
END_IF;

(* Alarm management *)
(* Position error *)
PositionErrorDelay(
	IN:= API.Activated AND API.Deactivated OR NOT (API.Activated OR API.Deactivated),
	PT:= init.PositionErrorDelay,
	Q  => API.PositionError);

(* Communicate status to HMI *)	
HMI := API;


 
          
END_FUNCTION_BLOCK

FUNCTION_BLOCK DutyStandbyClass
  VAR_INPUT
    Init : DutyStandbyClassInit_Typ;
    IO_IN : DutyStandbyClassIO_IN_Typ;
    API_IN : DutyStandbyClassAPI_IN_Typ;
  END_VAR
  VAR_OUTPUT
    IO_OUT : DutyStandbyClassIO_OUT_Typ;
    API_OUT : DutyStandbyClassAPI_OUT_Typ;
  END_VAR
  VAR
    Pump1 : BistableControlClass;
    Pump2 : BistableControlClass;
  END_VAR

            
          
END_FUNCTION_BLOCK

FUNCTION_BLOCK TankControlClass
  VAR_INPUT
    Init : TankControlClassInit_Typ;
    IO_IN : TankControlClassIO_IN_Typ;
    API_IN : TankControlClassAPI_IN_Typ;
  END_VAR
  VAR_OUTPUT
    IO_OUT : TankControlClassIO_OUT_Typ;
    API_OUT : TankControlClassAPI_OUT_Typ;
  END_VAR
  VAR
    DrainValve : BistableControlClass;
    FillingValve : BistableControlClass;
  END_VAR

            (* Description *)
(*Configure subclasses*)
DrainValve.init := Init.DrainValve;
FillingValve.init := Init.FillingValve;

(*Map inputs*)
DrainValve.io_in := IO_IN.DrainValve;
FillingValve.io_in := IO_IN.FillingValve;

(*Call the subclasses*)
DrainValve();
FillingValve();

(* Implement logic *)
API_OUT.TankLevel_pc := IO_IN.Level_cbm;

(*Map outputs*)
IO_OUT.DrainValve := DrainValve.io_out;
IO_OUT.FillingValve := FillingValve.io_out;
          
END_FUNCTION_BLOCK

FUNCTION_BLOCK ThreeWayIncrementValve
  VAR_INPUT
    ForwardCMD : BOOL;
    BackwardCMD : BOOL;
    cfgTaskSeq_ms : REAL;
    cfgOpenSpeed_s : REAL;
    cfgCloseSpeed_s : REAL;
  END_VAR
  VAR_OUTPUT
    Position : REAL := 0;
  END_VAR

            IF ForwardCMD AND NOT (Position >= 180) THEN
	Position := Position + (cfgOpenSpeed_s/cfgTaskSeq_ms);
ELSIF BackwardCMD AND NOT (Position <= -180) THEN
	Position := Position - (cfgCloseSpeed_s/cfgTaskSeq_ms);	
END_IF
          
END_FUNCTION_BLOCK

FUNCTION_BLOCK TwoWayIncrementValve
  VAR_INPUT
    OpenCMD : BOOL;
    CloseCMD : BOOL;
    cfgTaskSeq_ms : REAL;
    cfgOpenSpeed_s : REAL;
    cfgCloseSpeed_s : REAL;
  END_VAR
  VAR_OUTPUT
    Position : REAL := 0;
  END_VAR

            IF OpenCMD AND NOT (Position > 100) THEN
	Position := Position + (cfgOpenSpeed_s/cfgTaskSeq_ms);
ELSIF CloseCMD AND NOT (Position <= 0) THEN
	Position := Position - (cfgCloseSpeed_s/cfgTaskSeq_ms);	
END_IF
          
END_FUNCTION_BLOCK

FUNCTION_BLOCK fbAI_IF
  VAR_INPUT
    CFG : AI_CFG_Typ;  (* Configuration of the IO signal handler *)
    HW : REAL;  (* Connection to the AI card *)
  END_VAR
  VAR_OUTPUT
    SignalConn : AI_IO_Typ;  (* Connection to the global variable signal *)
  END_VAR

            SignalConn.PV := HW * CFG.Scale; (*Need to map*)
          
END_FUNCTION_BLOCK

FUNCTION_BLOCK fbAO_IF
  VAR_INPUT
    CFG : AO_CFG_Typ;  (* Configuration of the IO signal handler *)
    SignalConn : AO_IO_Typ;  (* Connection to the global variable signal *)
  END_VAR
  VAR_OUTPUT
    HW : REAL;  (* Connection to the AO card *)
  END_VAR

            HW := SignalConn.PV * CFG.Scale;
          
END_FUNCTION_BLOCK

FUNCTION_BLOCK fbDI_IF
  VAR_INPUT
    CFG : DI_CFG_Typ;  (* Configuration of the IO signal handler *)
    HW : BOOL;  (* Connection to the DI card *)
  END_VAR
  VAR_OUTPUT
    SignalConn : DI_IO_Typ;  (* Connection to the global variable signal *)
  END_VAR

            SignalConn.PV := HW;
          
END_FUNCTION_BLOCK

FUNCTION_BLOCK fbDO_IF
  VAR_INPUT
    CFG : DO_CFG_Typ;  (* Configuration of the IO signal handler *)
    SignalConn : DO_IO_Typ;  (* Connection to the global variable signal *)
  END_VAR
  VAR_OUTPUT
    HW : BOOL;  (* Connection to the DO card *)
  END_VAR

            HW := SignalConn.PV;
          
END_FUNCTION_BLOCK

FUNCTION_BLOCK Motor_Model
  VAR_INPUT
    CBActivated : BOOL := FALSE;
    LineVoltage : REAL := 440;
    cfgNominalPower : REAL := 12;  (* kW *)
    cfgPowerFactor : REAL := 0.83;
    Frequency : REAL := 60;
    cfgNoOfPoles : DINT := 4;
    cfgSpeedUpRate : REAL := 800;
    cfgSpeedDownRate : REAL := 800;
    simShortCircuit : BOOL := FALSE;
  END_VAR
  VAR_OUTPUT
    CurrentL1 : LREAL := 0;
    CurrentL2 : LREAL := 0;
    CurrentL3 : LREAL := 0;
    Speed : REAL := 0;
    Status : ARRAY[0..10] OF BOOL;
  END_VAR
  VAR
    vNs : REAL;
    vPhaseCurrent : REAL := 0;
    SpeedRamp : RAMP_REAL;
    SpeedBlink : BLINK;
    vBlinkTime : REAL;
    vBlinker : BOOL;
    vApparentPower_kVA : REAL;
  END_VAR

            Status[0] := CBActivated;;

vApparentPower_kVA := cfgNominalPower/(3*cfgPowerFactor);

vPhaseCurrent := (vApparentPower_kVA*1000)/LineVoltage;

CurrentL1 := (vPhaseCurrent/SQRT(3)+(BOOL_TO_REAL(simShortCircuit)*250))*BOOL_TO_REAL(Status[0]);
CurrentL2 := (vPhaseCurrent/SQRT(3)+(BOOL_TO_REAL(simShortCircuit)*250))*BOOL_TO_REAL(Status[0]);
CurrentL3 := (vPhaseCurrent/SQRT(3)+(BOOL_TO_REAL(simShortCircuit)*250))*BOOL_TO_REAL(Status[0]);

vNs := ((120 *Frequency)/DINT_TO_REAL(cfgNoOfPoles))*BOOL_TO_REAL(Status[0]);

SpeedRamp(
	IN:= vNs, 
	ASCEND:= cfgSpeedUpRate, 
	DESCEND:= cfgSpeedDownRate, 
	TIMEBASE:= T#2S, 
	OUT=>Speed);
	
vBlinkTime := 100000/MAX(1,Speed);

SpeedBlink(ENABLE:= vBlinkTime < 100000, TIMELOW:= REAL_TO_TIME(vBlinkTime), TIMEHIGH:= REAL_TO_TIME(vBlinkTime), OUT=> Status[1]);
          
END_FUNCTION_BLOCK

FUNCTION_BLOCK OnOffValve_Model
  VAR_INPUT
    OpenCmd : BOOL;  (* Command to open the valve *)
    CloseCmd : BOOL;  (* Command to close the valve *)
    cfgOpeningTime : TIME := TIME#5s0ms;  (* Time it take to open the valve *)
    cfgClosingTime : TIME := TIME#5s0ms;  (* Time it take to close the valve *)
    simOpenFail : BOOL;  (* Simulated open fail when true *)
    simCloseFail : BOOL;  (* Simulated close fail when true *)
  END_VAR
  VAR_OUTPUT
    Opened : BOOL;
    Closed : BOOL;
  END_VAR
  VAR
    OpenTime : TON;
    CloseTime : TON;
  END_VAR

            (* Description of action:
If the open/close signal comes the valve opens/closes in designated time *)

OpenTime(IN:= OpenCmd AND NOT Opened, PT:=cfgOpeningTime);
CloseTime(IN:= CloseCmd AND NOT Closed, PT:=cfgClosingTime);

IF Opened AND CloseCmd THEN
	Opened := FALSE;
ELSIF OpenTime.Q AND NOT simOpenFail THEN
	Opened := TRUE;
END_IF

IF Closed AND OpenCmd THEN
	Closed := FALSE;
ELSIF CloseTime.Q AND NOT simCloseFail THEN
	Closed := TRUE;
END_IF
          
END_FUNCTION_BLOCK

FUNCTION_BLOCK Pump_Model
  VAR_INPUT
    OnCmd : BOOL;  (* Pump simulator will turn on when recieves ON signal and will shutoff when it recieves a OFF signal If SimTrip signal becomes true, pump will trip and cannot be started until signal goes false If SimFilterFail signal becomes true the pump will operate but the flowrate will start to slowly drop until zero *)
    OffCmd : BOOL;
    SimTrip : BOOL := FALSE;
    SimFilterFail : BOOL := FALSE;
    NoWater : BOOL := FALSE;  (* This tells the pump simulation that there is no more medium to pump so the flowmeter drops to 0 *)
    cfgFlowrate : REAL := 3000;
    cfgRampUpRate : REAL := 150;
    cfgRampDownRate : REAL := 150;
  END_VAR
  VAR_OUTPUT
    RunStatus : DINT;  (* 0 - Stopped, 1 - Running *)
    FlowmeterOut : REAL;  (* Cubic meters per hour *)
  END_VAR
  VAR
    PumpSR : SR;
    vPumpRunning : BOOL;
    Flowmeter : RAMP_REAL;
    vFlowmeterSP : REAL;
    vAscend : REAL;
    vDescend : REAL;
  END_VAR

            
PumpSR(SET1:= OnCmd AND NOT (OffCmd OR SimTrip OR RunStatus=1) , RESET:= (OffCmd OR SimTrip), Q1=>vPumpRunning );

RunStatus := BOOL_TO_DINT(vPumpRunning);

IF vPumpRunning AND NOT NoWater THEN
	vFlowmeterSP := BOOL_TO_REAL( NOT SimFilterFail) * cfgFlowrate;
	vAscend := cfgRampUpRate;
	vDescend := cfgRampDownRate;
ELSE
	vFlowmeterSP := 0;
	vAscend := 0;
	vDescend := 99999999;
END_IF


Flowmeter(
	IN:= vFlowmeterSP, 
	ASCEND:= vAscend,
	TIMEBASE:= T#500MS, 
	DESCEND:= vDescend, 
	OUT=> FlowmeterOut);
          
END_FUNCTION_BLOCK

FUNCTION_BLOCK Tank_Model
  VAR_INPUT
    cfgTaskCycle : REAL;  (* Task cycle of the POU this model is running in miliseconds *)
    cfgLenght : REAL := 0;  (* Lenght of the tank in meters *)
    cfgWidth : REAL := 0;  (* Width of the tank in meters *)
    cfgHeight : REAL := 0;  (* Height of the tank in meters *)
    cfgStartLevel : REAL := 0;  (* Starting level of the tank in m~3 *)
    cfgFSHH : REAL := 95;  (* Float switch high high level in percentages of the volume of the tank *)
    cfgFSH : REAL := 80;  (* Float switch high level in percentages of the volume of the tank *)
    cfgFSL : REAL := 20;  (* Float switch low level in percentages of the volume of the tank *)
    cfgFSLL : REAL := 5;  (* Float switch low low level in percentages of the volume of the tank *)
    Inflow1 : REAL := 0;  (* Inflow, slot 1 to the tank in cubic meters per hour *)
    Inflow2 : REAL := 0;  (* Inflow, slot 2 to the tank in cubic meters per hour *)
    Inflow3 : REAL := 0;  (* Inflow, slot 3 to the tank in cubic meters per hour *)
    Inflow4 : REAL := 0;  (* Inflow, slot 4 to the tank in cubic meters per hour *)
    Inflow5 : REAL := 0;  (* Inflow, slot 5 to the tank in cubic meters per hour *)
    Outflow1 : REAL := 0;  (* Outflow, slot 1 to the tank in cubic meters per hour *)
    Outflow2 : REAL := 0;  (* Outflow, slot 2 to the tank in cubic meters per hour *)
    Outflow3 : REAL := 0;  (* Outflow, slot 3 to the tank in cubic meters per hour *)
    Outflow4 : REAL := 0;  (* Outflow, slot 4 to the tank in cubic meters per hour *)
    Outflow5 : REAL := 0;  (* Outflow, slot 5 to the tank in cubic meters per hour *)
  END_VAR
  VAR_OUTPUT
    TankLevel_cbm : REAL;  (* Tank level in cubic meters *)
    TankLevel_pc : REAL;  (* Tank level in percentages *)
    FSHHActive : BOOL;  (* Floating switch High high level active *)
    FSHActive : BOOL;  (* Floating switch High level active *)
    FSLActive : BOOL;  (* Floating switch Low level active *)
    FSLLActive : BOOL;  (* Floating switch Low low level active *)
  END_VAR
  VAR
    vNominalVolume : REAL;
    vInflowTotal : REAL;
    vOutflowTotal : REAL;
    vDeltaTime : REAL;
  END_VAR
  VAR RETAIN
    vColdRestart : BOOL;
  END_VAR

            IF NOT vColdRestart THEN
	TankLevel_cbm := cfgStartLevel;
	vColdRestart := TRUE;
END_IF

vNominalVolume := cfgLenght * cfgWidth * cfgHeight;

vInflowTotal := Inflow1 + Inflow2 + Inflow3 + Inflow4 + Inflow5;

vOutflowTotal := Outflow1 + Outflow2 + Outflow3 + Outflow4 + Outflow5;

(* Task cycle speed increase will lower the speed of TankLevel filling *)
vDeltaTime := cfgTaskCycle/DINT_TO_REAL(3600 * 1000);

(* Tank level calculation, independent of task execution cycle *)
TankLevel_cbm :=LIMIT(0,TankLevel_cbm + (vInflowTotal - vOutflowTotal) * vDeltaTime, vNominalVolume);

TankLevel_pc := (TankLevel_cbm / vNominalVolume) * 100;

(* Limit switch handling *)
FSHHActive := TankLevel_pc >= cfgFSHH;
FSHActive := TankLevel_pc >= cfgFSH;
FSLActive := TankLevel_pc <= cfgFSL;
FSLLActive := TankLevel_pc <= cfgFSLL;
          
END_FUNCTION_BLOCK

FUNCTION_BLOCK WorkplaceHandle
  VAR_INPUT
    WorkplaceIn : ARRAY[0..20] OF BOOL;  (* 0 System theme button, 1-7 Buttons 1-7 *)
    Button1Txt : STRING := 'Button1';  (* Text for workplace button 1 *)
    Button2Txt : STRING := 'Button2';  (* Text for workplace button 2 *)
    Button3Txt : STRING := 'Button3';  (* Text for workplace button 3 *)
    Button4Txt : STRING := 'Button4';  (* Text for workplace button 4 *)
    Button5Txt : STRING := 'Button5';  (* Text for workplace button 5 *)
    Button6Txt : STRING := 'Button6';  (* Text for workplace button 6 *)
    Button7Txt : STRING := 'Button7';  (* Text for workplace button 7 *)
    Button8Txt : STRING := 'Button8';  (* Text for workplace button 8 *)
    Button9Txt : STRING := 'Button9';  (* Text for workplace button 9 *)
    NavBarFillColor1 : DWORD := 16#FF097500;  (* RGB hex code string for navigation bar color *)
    NavBarFrameColor1 : DWORD := 16#FF000000;  (* RGB hex code string for navigation bar frame color *)
    NavBarFillColor2 : DWORD := 16#FF002B06;  (* RGB hex code string for navigation bar color *)
    NavBarFrameColor2 : DWORD := 16#FF000000;  (* RGB hex code string for navigation bar frame color *)
    ButtonsColor1 : DWORD := 16#FF777777;  (* RGB hex code for buttons color 1 *)
    ButtonsColor2 : DWORD := 16#FF232323;  (* RGB hex code for buttons color 2 *)
    StatusBarFillColor1 : DWORD := 16#FF000000;  (* RGB hex code for status bar *)
    StatusBarFrameColor1 : DWORD := 16#FF000000;  (* RGB hex code for status bar *)
    StatusBarFillColor2 : DWORD := 16#FF000000;  (* RGB hex code for status bar *)
    StatusBarFrameColor2 : DWORD := 16#FF000000;  (* RGB hex code for status bar *)
    ProjectName : STRING := 'TKAutomation project';  (* Project name *)
    NoOfVisibleButtons : DINT := 9;  (* Number of visible buttons. Max 9 *)
  END_VAR
  VAR_OUTPUT
    WorkplaceText : ARRAY[0..20] OF STRING;  (* Project name, 1-9 Button text *)
    WorkplaceOut : ARRAY[0..20] OF DINT;  (* 0 - ScreenSelected, 1 - Visible buttons *)
    WorkplaceColor : ARRAY[0..20] OF DWORD;  (* 0 - NavBarFillColor, 1 - NavBarFrameColor, 2 - ButtonsColor1, 3 - ButtonsColor2, 4 - StatusBarFillColor, 5 - StatusBarFrameColor *)
  END_VAR

            (* Menu selector buttons bit 1 - 9 *)
IF WorkplaceIn[1] THEN
	WorkplaceOut[0] := 0;
END_IF
IF WorkplaceIn[2] THEN
	WorkplaceOut[0] := 1;
END_IF
IF WorkplaceIn[3] THEN
	WorkplaceOut[0] := 2;
END_IF
IF WorkplaceIn[4] THEN
	WorkplaceOut[0] := 3;
END_IF
IF WorkplaceIn[5] THEN
	WorkplaceOut[0] := 4;
END_IF
IF WorkplaceIn[6] THEN
	WorkplaceOut[0] := 5;
END_IF
IF WorkplaceIn[7] THEN
	WorkplaceOut[0] := 6;
END_IF
IF WorkplaceIn[8] THEN
	WorkplaceOut[0] := 7;
END_IF
IF WorkplaceIn[9] THEN
	WorkplaceOut[0] := 8;
END_IF

(* Bit 1 - System theme *)
WorkplaceOut[1]:= BOOL_TO_DINT(WorkplaceIn[0]);
WorkplaceOut[2]:= NoOfVisibleButtons;

WorkplaceText[0] := ProjectName;
WorkplaceText[1] := Button1Txt;
WorkplaceText[2] := Button2Txt;
WorkplaceText[3] := Button3Txt;
WorkplaceText[4] := Button4Txt;
WorkplaceText[5] := Button5Txt;
WorkplaceText[6] := Button6Txt;
WorkplaceText[7] := Button7Txt;
WorkplaceText[8] := Button8Txt;
WorkplaceText[9] := Button9Txt;

WorkplaceColor[0]:= NavBarFillColor1;
WorkplaceColor[1]:= NavBarFrameColor1;
WorkplaceColor[2]:= NavBarFillColor2;
WorkplaceColor[3]:= NavBarFrameColor2;
WorkplaceColor[4]:= ButtonsColor1;
WorkplaceColor[5]:= ButtonsColor2;
WorkplaceColor[6]:= StatusBarFillColor1;
WorkplaceColor[7]:= StatusBarFrameColor1;
WorkplaceColor[8]:= StatusBarFillColor2;
WorkplaceColor[9]:= StatusBarFrameColor2;




          
END_FUNCTION_BLOCK

PROGRAM Main
  VAR
    FWStorageTank : TankControlClass;  (* Control system of the Fresh water storage tank *)
    FWServiceTank : TankControlClass;  (* Control system of the Fresh water service tank *)
    FWFeedControl : DutyStandbyClass;  (* Control class of the Feed pumps, provides automatic start/stop and fault recovery *)
    HFOFuelHeatingValve : BistableControlClass;  (* Valve controlling the steam towards HFO fuel heating system *)
    HVACSystemValve : BistableControlClass;  (* Valve controlling the steam towards HVAC system *)
    OperationalConsumersValve : BistableControlClass;  (* Valve controlling the steam towards Operational consumers *)
    SteamDumpValve : BistableControlClass;  (* Valve controlling the steam when consumers are not consuming enough steam *)
    ReliefValve : BistableIndicationClass;  (* Indication that the relief valve has triggered *)
    BurnerControl : BurnerControlClass;  (* Class controlling the burner system and steam production *)
  END_VAR

                    (* Main program using actions to section code *)
MapInputs();

FWTankSystem();
SteamConsumerSystem();

MapOutputs();

                  

ACTION FWTankSystem:
                        (***Fresh water tank system control and monitoring***)
(*Requirements:
- Needs to regulate fresh water storage tank level
- Needs to refill fresh water storage tank level with a FWStorageTankFillingValve
- All tanks need to be able to drain water into collecting tank/outside of the ship
- Service tank needs to regulate the tank level to a specific level to optimize steam production, this is to be configurable
- Service tank needs to be drained into collecting tank/outside of the ship
- FWFeed pumps will work with the duty change over, change over occurs on demand by the operator or by a fault in the device
- Changeover is only if pumps are in automatic mode, other mode is manual
- FWFeed pumps pump water from the storage tank to the service tank*)

(* Instantiate classes *)
//FRESH WATER STORAGE TANK
FWStorageTank();

//SERVICE TANK
FWServiceTank();

//Duty standby pumps
FWFeedControl();

(* Automatic control *)
                      
END_ACTION

ACTION SteamConsumerSystem:
                        (* This system controls the steam valves to the consumers *)
(*Requirements:
- Operator needs to be able to open and close any valve on the consumer system
- The consumer valves are only in manual mode
- The valves need to be open incrementally
*)

                      
END_ACTION

ACTION SteamProductionSystem:
                        
                      
END_ACTION

ACTION MapInputs:
                        (*Map inputs of the FW Service tank *)
FWStorageTank.IO_IN.DrainValve.Activated := IO.DIS.x200_FW_STORAGE_TK_DRAINVALVE_CLOSED.PV;
FWStorageTank.IO_IN.DrainValve.Deactivated := IO.DIS.x200_FW_STORAGE_TK_DRAINVALVE_OPENED.PV;
FWStorageTank.IO_IN.DrainValve.ReadyToOperate := IO.DIS.x200_FW_STORAGE_TK_DRAINVALVE_READY.PV;
FWStorageTank.IO_IN.DrainValve.Remote := IO.DIS.x200_FW_STORAGE_TK_DRAINVALVE_REMOTE.PV;
FWStorageTank.IO_IN.DrainValve.Tripped := FALSE;

FWStorageTank.IO_IN.FillingValve.Activated := IO.DIS.x200_FW_STORAGE_TK_FILLVALVE_CLOSED.PV;
FWStorageTank.IO_IN.FillingValve.Deactivated := IO.DIS.x200_FW_STORAGE_TK_FILLVALVE_OPENED.PV;
FWStorageTank.IO_IN.FillingValve.ReadyToOperate := IO.DIS.x200_FW_STORAGE_TK_FILLVALVE_READY.PV;
FWStorageTank.IO_IN.FillingValve.Remote := IO.DIS.x200_FW_STORAGE_TK_FILLVALVE_REMOTE.PV;
FWStorageTank.IO_IN.FillingValve.Tripped := FALSE;

FWStorageTank.IO_IN.HLimitSwitch := IO.DIS.x200_FW_STORAGE_TK_HLIMITSWITCH.PV;
FWStorageTank.IO_IN.LLimitSwitch := IO.DIS.x200_FW_STORAGE_TK_LLIMITSWITCH.PV;

FWStorageTank.IO_IN.Level_cbm := IO.AIS.x200_FRESH_WATER_STORAGE_TANK_LEVEL.PV;

(*Map inputs of the FW service tank*)
FWServiceTank.IO_IN.DrainValve.Activated := IO.DIS.x200_FW_SERVICE_TK_DRAINVALVE_CLOSED.PV;
FWServiceTank.IO_IN.DrainValve.Deactivated := IO.DIS.x200_FW_SERVICE_TK_DRAINVALVE_OPENED.PV;
FWServiceTank.IO_IN.DrainValve.ReadyToOperate := IO.DIS.x200_FW_SERVICE_TK_DRAINVALVE_READY.PV;
FWServiceTank.IO_IN.DrainValve.Remote := IO.DIS.x200_FW_SERVICE_TK_DRAINVALVE_REMOTE.PV;
FWServiceTank.IO_IN.DrainValve.Tripped := FALSE;

FWServiceTank.IO_IN.FillingValve.Activated := IO.DIS.x200_FW_SERVICE_TK_FILLVALVE_CLOSED.PV;
FWServiceTank.IO_IN.FillingValve.Deactivated := IO.DIS.x200_FW_SERVICE_TK_FILLVALVE_OPENED.PV;
FWServiceTank.IO_IN.FillingValve.ReadyToOperate := IO.DIS.x200_FW_SERVICE_TK_FILLVALVE_READY.PV;
FWServiceTank.IO_IN.FillingValve.Remote := IO.DIS.x200_FW_SERVICE_TK_FILLVALVE_REMOTE.PV;
FWServiceTank.IO_IN.FillingValve.Tripped := FALSE;

FWServiceTank.IO_IN.HLimitSwitch := IO.DIS.x200_FW_SERVICE_TK_HLIMITSWITCH.PV;
FWServiceTank.IO_IN.LLimitSwitch := IO.DIS.x200_FW_SERVICE_TK_LLIMITSWITCH.PV;

FWServiceTank.IO_IN.Level_cbm := IO.AIS.x200_FRESH_WATER_SERVICE_TANK_LEVEL.PV;

(*Map inputs of the FW feed control *)
FWFeedControl.IO_IN.Pump1.Activated := IO.DIS.x200_FW_SERVICE_PUMP1_RUNNING.PV;
FWFeedControl.IO_IN.Pump1.Deactivated := IO.DIS.x200_FW_SERVICE_PUMP1_STOPPED.PV;
FWFeedControl.IO_IN.Pump1.ReadyToOperate := IO.DIS.x200_FW_SERVICE_PUMP1_READY.PV;
FWFeedControl.IO_IN.Pump1.Remote := IO.DIS.x200_FW_SERVICE_PUMP1_REMOTE.PV;
FWFeedControl.IO_IN.Pump1.Tripped := IO.DIS.x200_FW_SERVICE_PUMP1_TRIPPED.PV;

FWFeedControl.IO_IN.Pump2.Activated := IO.DIS.x200_FW_SERVICE_PUMP2_RUNNING.PV;
FWFeedControl.IO_IN.Pump2.Deactivated := IO.DIS.x200_FW_SERVICE_PUMP2_STOPPED.PV;
FWFeedControl.IO_IN.Pump2.ReadyToOperate := IO.DIS.x200_FW_SERVICE_PUMP2_READY.PV;
FWFeedControl.IO_IN.Pump2.Remote := IO.DIS.x200_FW_SERVICE_PUMP2_REMOTE.PV;
FWFeedControl.IO_IN.Pump2.Tripped := IO.DIS.x200_FW_SERVICE_PUMP2_TRIPPED.PV;
                      
END_ACTION

ACTION MapOutputs:
                        (*FW Storage tank outputs*)
IO.DOS.x200_FW_STORAGE_TANK_DRAINVALVE_CLOSECMD.PV := FWStorageTank.IO_OUT.DrainValve.ActivateCmd; 
IO.DOS.x200_FW_STORAGE_TANK_DRAINVALVE_OPENCMD.PV := FWStorageTank.IO_OUT.DrainValve.DeactivateCmd;
IO.DOS.x200_FW_STORAGE_TANK_FILLVALVE_CLOSECMD.PV := FWStorageTank.IO_OUT.FillingValve.ActivateCmd; 
IO.DOS.x200_FW_STORAGE_TANK_FILLVALVE_OPENCMD.PV := FWStorageTank.IO_OUT.FillingValve.DeactivateCmd;

(*FW Service tank outputs*)
IO.DOS.x200_FW_SERVICE_TANK_DRAINVALVE_CLOSECMD.PV := FWServiceTank.IO_OUT.DrainValve.ActivateCmd; 
IO.DOS.x200_FW_SERVICE_TANK_DRAINVALVE_OPENCMD.PV := FWServiceTank.IO_OUT.DrainValve.DeactivateCmd;
IO.DOS.x200_FW_SERVICE_TANK_FILLVALVE_CLOSECMD.PV := FWServiceTank.IO_OUT.FillingValve.ActivateCmd; 
IO.DOS.x200_FW_SERVICE_TANK_FILLVALVE_OPENCMD.PV := FWServiceTank.IO_OUT.FillingValve.DeactivateCmd;

(*FW Feed control outputs*)
IO.DOS.x200_FW_SERVICE_PUMP1_STARTCMD.PV := FWFeedControl.IO_OUT.Pump1.ActivateCmd;
IO.DOS.x200_FW_SERVICE_PUMP1_STOPCMD.PV := FWFeedControl.IO_OUT.Pump1.DeactivateCmd;

IO.DOS.x200_FW_SERVICE_PUMP2_STARTCMD.PV := FWFeedControl.IO_OUT.Pump2.ActivateCmd;
IO.DOS.x200_FW_SERVICE_PUMP2_STOPCMD.PV := FWFeedControl.IO_OUT.Pump2.DeactivateCmd;
                      
END_ACTION
END_PROGRAM

PROGRAM Workplace
  VAR
    vPositionMsg : STRING;
    vFWServiceTankMsg : STRING;
    vFWStorageTankMsg : STRING;
  END_VAR

                    // (* Workplace handle call *)
// WorkplaceCall(
// 	WorkplaceIn:= vWorkplaceIn, 
// 	Button1Txt:= 'Main', 
// 	Button2Txt:= 'Config', 
// 	Button3Txt:= 'Graphs', 
// 	Button4Txt:= 'Alarms', 
// 	ProjectName:= 'Automation of Ships Steam Boiler' , 
// 	NoOfVisibleButtons:= 4, 
// 	WorkplaceText=> vWorkplaceText, 
// 	WorkplaceOut=> vWorkplaceOut,
// 	WorkplaceColor=>vWorkplaceColor);
// 
// (* Graphic element visibility *)
// vAutoStartVisible := GVL.IO_Typ.DIS_Typ.RemoteSW AND NOT GVL.LIO.ResetRequired AND GVL.LIO.IgnitionSeq = 1;
// vManStartVisible := NOT GVL.IO_Typ.DIS_Typ.RemoteSW AND NOT GVL.LIO.ResetRequired AND GVL.LIO.IgnitionSeq = 1;
// vLoadUpVisible := NOT GVL.IO_Typ.DIS_Typ.RemoteSW AND GVL.LIO.IgnitionSeq = 4;
// vLoadDownVisible := NOT GVL.IO_Typ.DIS_Typ.RemoteSW AND GVL.LIO.IgnitionSeq = 4;
// vResetButtonVisible := GVL.LIO.ResetRequired;
// vIgniteButtonVisible := NOT GVL.IO_Typ.DIS_Typ.RemoteSW AND GVL.LIO.IgnitionSeq = 3;
// vAutoStopButtonVisible := GVL.IO_Typ.DIS_Typ.RemoteSW AND GVL.LIO.IgnitionSeq <> 12;
// vManStopButtonVisible := NOT GVL.IO_Typ.DIS_Typ.RemoteSW AND GVL.LIO.IgnitionSeq <> 12;
// vFlameVisible := GVL.LIO.FlameEstablished;
// vSteamPipeActive := GVL.IO_Typ.AIS_Typ.SteamPressure > 0;
// vCondensatePipeActive := GVL.LIO.SteamCondensation > 0;
// vFWPP1Master := GVL.LIO.MasterFWPP = 1;
// vFWPP2Master := GVL.LIO.MasterFWPP = 2;
// vFlowToFWTk := (GVL.IO_Typ.AOS_Typ.FWTkRegValve > 0) AND (GVL.IO_Typ.DOS_Typ.FWPump1 OR GVL.IO_Typ.DOS_Typ.FWPump2);
// vSteamDumpActive := vSteamPipeActive AND (GVL.LIO.SteamDump > 0);
// vFuelPipeActive := GVL.IO_Typ.DIS_Typ.MainFuelValveOpen;
// vSystemLoad := GVL.LIO.SteamConsumers;
// vAirOpen := LIMIT(0,REAL_TO_INT(GVL.IO_Typ.AOS_Typ.AirValve/5) , 20);
// 
// 
// IF GVL.IO_Typ.DIS_Typ.RemoteSW THEN
// 	vPositionMsg := GVL.CFG_Typ.TxtRemote;
// ELSE
// 	vPositionMsg := GVL.CFG_Typ.TxtManual;
// END_IF
// 
// IF GVL.IO_Typ.AIS_Typ.FWTank_Level >=GVL.CFG_Typ.FWTankHighLimit THEN
// 	vFWServiceTankMsg := GVL.CFG_Typ.TxtOvrFl;
// ELSIF GVL.IO_Typ.AIS_Typ.FWTank_Level <= GVL.CFG_Typ.FWTankLowLimit THEN
// 	vFWServiceTankMsg := GVL.CFG_Typ.TxtFWTkEmpty;
// ELSE
// 	vFWServiceTankMsg := 'FW Service Tank';
// END_IF
// 
// IF GVL.IO_Typ.AIS_Typ.FWSTORETank_Level >=GVL.CFG_Typ.FWTankHighLimit THEN
// 	vFWServiceTankMsg := GVL.CFG_Typ.TxtOvrFl;
// ELSIF GVL.IO_Typ.AIS_Typ.FWSTORETank_Level <= GVL.CFG_Typ.FWTankLowLimit THEN
// 	vFWStorageTankMsg := GVL.CFG_Typ.TxtFWTkEmpty;
// ELSE
// 	vFWStorageTankMsg := 'FW Storage Tank';
// END_IF
                  
END_PROGRAM

PROGRAM Simulator
  VAR
    FWServiceTank : Tank_Model;
    FWStorageTank : Tank_Model;
  END_VAR

                    (*FW System simulation*)
FWSystemSIM();

// (* Valve open/close simulation *)
// 
// MainFuelValve(
// 	OpenCmd:= GVL.IO.DOS.FuelValveOpenCmd, 
// 	CloseCmd:= GVL.IO.DOS.FuelValveCloseCmd, 
// 	cfgOpeningTime:= GVL.SimCFG.ValveOperatingTime, 
// 	cfgClosingTime:= GVL.SimCFG.ValveOperatingTime, 
// 	simOpenFail:= vFVOpenFail, 
// 	simCloseFail:= vFVCloseFail, 
// 	Opened=> GVL.IO.DIS.MainFuelValveOpen , 
// 	Closed=> GVL.IO.DIS.MainFuelValveClosed );
// 	
// HFOHeatValve(
// 	OpenCmd:= GVL.IO.DOS.HFOHeatValveOpenCmd, 
// 	CloseCmd:= GVL.IO.DOS.HFOHeatValveCloseCmd, 
// 	cfgOpeningTime:= GVL.SimCFG.ValveOperatingTime, 
// 	cfgClosingTime:= GVL.SimCFG.ValveOperatingTime, 
// 	simOpenFail:= vHFOpenFail, 
// 	simCloseFail:= vHFOCloseFail, 
// 	Opened=> GVL.IO.DIS.HFOHeatValveOpen, 
// 	Closed=> GVL.IO.DIS.HFOHeatValveClosed);
// 
// HVACHeatValve(
// 	OpenCmd:= GVL.IO.DOS.HVACHeatValveOpenCmd, 
// 	CloseCmd:= GVL.IO.DOS.HVACHeatValveCloseCmd, 
// 	cfgOpeningTime:= GVL.SimCFG.ValveOperatingTime, 
// 	cfgClosingTime:= GVL.SimCFG.ValveOperatingTime, 
// 	simOpenFail:= vHVACOpenFail, 
// 	simCloseFail:= vHVACCloseFail, 
// 	Opened=> GVL.IO.DIS.HVACHeatValveOpen, 
// 	Closed=> GVL.IO.DIS.HVACHeatValveClosed);
// 
// OperConsValve(
// 	OpenCmd:= GVL.IO.DOS.OperConsValveOpenCmd, 
// 	CloseCmd:= GVL.IO.DOS.OperConsValveCloseCmd, 
// 	cfgOpeningTime:= GVL.SimCFG.ValveOperatingTime, 
// 	cfgClosingTime:= GVL.SimCFG.ValveOperatingTime, 
// 	simOpenFail:= vOperConsOpenFail, 
// 	simCloseFail:= vOperConsCloseFail, 
// 	Opened=> GVL.IO.DIS.OperConsValveOpen, 
// 	Closed=> GVL.IO.DIS.OperConsValveClosed);
// 	
// (* Burner ignited, burning*)
// IF GVL.IO.AOS.FuelValve > 0 
// 	AND (GVL.IO.DOS.Ignitor OR vFlameEstablished)
// 	AND GVL.IO.DIS.MainFuelValveOpen THEN
// 	vFlameEstablished := TRUE;
// ELSE
// 	vFlameEstablished := FALSE;
// END_IF
// 
// Photocell1DetectDelay(IN:= vFlameEstablished, PT:=GVL.SimCFG.PCell1DetectDelay);
// Photocell2DetectDelay(IN:= vFlameEstablished, PT:=GVL.SimCFG.PCell2DetectDelay);
// 
// GVL.IO.DIS.Photocell1 := Photocell1DetectDelay.Q AND NOT vPhotocell1Dirty;
// GVL.IO.DIS.Photocell2 := Photocell1DetectDelay.Q AND NOT vPhotocell2Dirty;
// 
// (*Steam pressure production simulation*)
// (*Steam consumer simulation*)
// 
// GVL.IO.AIS.HFOHeatingConsumer := BOOL_TO_REAL(GVL.IO.DIS.HFOHeatValveOpen)*vHFOMultiplier * GVL.SysCFG.HFOConsumerNominal;
// 
// GVL.IO.AIS.HVACSystemConsumer := BOOL_TO_REAL(GVL.IO.DIS.HVACHeatValveOpen)*vHVACMultiplier * GVL.SysCFG.HVACConsumerNominal;
// 
// GVL.IO.AIS.OperationalConsumers := BOOL_TO_REAL(GVL.IO.DIS.OperConsValveOpen)*vOperMultiplier * GVL.SysCFG.OperConsumerNominal; 
// 
// vPressureRelief := MAX(0, GVL.IO.AIS.SteamPressure - GVL.SimCFG.ReliefValveOpeningSP);
// vRotateReliefValve := REAL_TO_DINT(LIMIT(0, 10*vPressureRelief, 180));
// 
// vSteamDump := 0.1 * GVL.IO.AOS.SteamDumpValve;
// 
// vSteamConsumers := GVL.IO.AIS.HFOHeatingConsumer
// 				 + GVL.IO.AIS.HVACSystemConsumer
// 				 + GVL.IO.AIS.OperationalConsumers
// 				 + vPressureRelief
// 				 + vSteamDump;
// 				 
// (* Steam producers *)
// vSteamProduction := (GVL.SimCFG.SteamFactor * GVL.IO.AOS.FuelValve 
// 					+ BOOL_TO_REAL(vOverpressurize)*GVL.SimCFG.OverpressureMultiplier)* BOOL_TO_REAL(vFlameEstablished);
// 					
// (* Water evaporation/condensation *)					
// vWaterEvaporation := GVL.SimCFG.WaterEvapFactor * vSteamProduction;
// 
// vLostWater := GVL.SimCFG.LostWaterOnConsumers * vSteamConsumers;
// vSteamCondensation := vWaterEvaporation;
// 
// GVL.IO.AIS.SteamPressure := LIMIT(0, GVL.IO.AIS.SteamPressure + vSteamProduction - vSteamConsumers, 9999);
// 
// 
// (* FW Pumps simulation *)
// FWServicePump1(
// 	OnCmd:= GVL.IO.DOS.FWPump1, 
// 	OffCmd:= NOT GVL.IO.DOS.FWPump1, 
// 	NoWater:= GVL.IO.AIS.FWSTORETank_Level <= 0, 
// 	cfgFlowrate:= 5000, 
// 	cfgRampUpRate:= 100, 
// 	cfgRampDownRate:= 100, 
// 	RunStatus=> GVL.IO.DIS.FWServicePump1, 
// 	FlowmeterOut=> vFWServicePump1Flow);
// 	
// FWServicePump2(
// 	OnCmd:= GVL.IO.DOS.FWPump2, 
// 	OffCmd:= NOT GVL.IO.DOS.FWPump2, 
// 	NoWater:= GVL.IO.AIS.FWSTORETank_Level <= 0, 
// 	cfgFlowrate:= 5000, 
// 	cfgRampUpRate:= 100, 
// 	cfgRampDownRate:= 100, 
// 	RunStatus=> GVL.IO.DIS.FWServicePump2, 
// 	FlowmeterOut=> vFWServicePump2Flow);
// 


// 				
// (* Blower spinning simulation *)
// SimBlink(ENABLE:=GVL.IO.DOS.AirBlowerMotor , TIMELOW:=GVL.SimCFG.BlinkFreq , TIMEHIGH:=GVL.SimCFG.BlinkFreq , OUT=>vBlink );
// 
// (* Send system information to other programs *)
// GVL.LIO.FlameEstablished := vFlameEstablished;
// GVL.LIO.SteamCondensation := vSteamCondensation;
// GVL.LIO.SteamDump := vSteamDump;
// GVL.LIO.SteamConsumers := vSteamConsumers;
                  

ACTION FWSystemSIM:
                        (*Water tanks simulation*)
//vServiceTankDrainFlow := 8000 * BOOL_TO_REAL(vDrainServiceTank);
//vFillStorageTankFlow := 8000 * BOOL_TO_REAL(vFillStorageTk);

(* FW Service Tk *)
FWServiceTank(
	cfgTaskCycle:= 200, 
	cfgLenght:= 5, 
	cfgWidth:= 5, 
	cfgHeight:= 7, 
	cfgFSHH:= 95, 
	cfgFSH:= 85, 
	cfgFSL:= 15, 
	cfgFSLL:= 5, 
	//Inflow1:= (GVL.IO.AOS.FWTkRegValve/100) * vFWServicePump1Flow, 
	//Inflow2:= (GVL.IO.AOS.FWTkRegValve/100) * vFWServicePump2Flow, 
	//Outflow1:= vWaterEvaporation*10000,
	//Outflow2:= vServiceTankDrainFlow, 
	TankLevel_pc=> IO.AIS.x200_FRESH_WATER_SERVICE_TANK_LEVEL.PV, 
	//FSHHActive=> GVL.IO.DIS.FWTankLSHighHigh , 
	FSHActive=> IO.DIS.x200_FW_SERVICE_TK_HLIMITSWITCH.PV, 
	FSLActive=> IO.DIS.x200_FW_SERVICE_TK_LLIMITSWITCH.PV
	//FSLLActive=> GVL.IO.DIS.FWTankLSLowLow
);
	
//vFWStorageInflow := vSteamCondensation*10000
				// + ((vFWServicePump1Flow + vFWServicePump2Flow)
					//- (GVL.IO.AOS.FWTkRegValve)/100 *(vFWServicePump1Flow + vFWServicePump2Flow)) ;	
FWStorageTank(
	cfgTaskCycle:= 200 , 
	cfgLenght:= 10, 
	cfgWidth:= 10, 
	cfgHeight:= 10, 
	cfgStartLevel := 800,
	//Inflow1:= vFWStorageInflow,
	//Inflow2:= vFillStorageTankFlow, 
	//Outflow1:= vFWServicePump1Flow, 
	//Outflow2:= vFWServicePump2Flow,
	//Outflow3:= vLostWater,
	TankLevel_pc=> IO.AIS.x200_FRESH_WATER_STORAGE_TANK_LEVEL.PV);
                      
END_ACTION
END_PROGRAM

PROGRAM AOS_POU
  VAR
    x150_BOILER_WATER_FEED_REGULATION_VALVE_SETPOINT : fbAO_IF := (CFG := (sigMin := 0, sigMax := 100, Scale := 1));  (* Signal conditioning module *)
    x150_STEAM_DUMP_VALVE_SETPOINT : fbAO_IF := (CFG := (sigMin := 0, sigMax := 100, Scale := 1));  (* Signal conditioning module *)
    x100_AIR_VALVE_SETPOINT : fbAO_IF := (CFG := (sigMin := 0, sigMax := 100, Scale := 1));  (* Signal conditioning module *)
    x100_FUEL_VALVE_SETPOINT : fbAO_IF := (CFG := (sigMin := 0, sigMax := 100, Scale := 1));  (* Signal conditioning module *)
  END_VAR

                    IF NOT GVL.SIMULATE THEN
(* Analog output signal conditioning function block call *)
x150_BOILER_WATER_FEED_REGULATION_VALVE_SETPOINT(SignalConn := IO.AOS.x150_BOILER_WATER_FEED_REGULATION_VALVE_SETPOINT);
x150_STEAM_DUMP_VALVE_SETPOINT(SignalConn := IO.AOS.x150_STEAM_DUMP_VALVE_SETPOINT);
x100_AIR_VALVE_SETPOINT(SignalConn := IO.AOS.x100_AIR_VALVE_SETPOINT);
x100_FUEL_VALVE_SETPOINT(SignalConn := IO.AOS.x100_FUEL_VALVE_SETPOINT);
END_IF

                  
END_PROGRAM

PROGRAM DOS_POU
  VAR
    x200_FW_SERVICE_PUMP1_STARTCMD : fbDO_IF;  (* Signal conditioning module *)
    x200_FW_SERVICE_PUMP1_STOPCMD : fbDO_IF;  (* Signal conditioning module *)
    x200_FW_SERVICE_PUMP2_STARTCMD : fbDO_IF;  (* Signal conditioning module *)
    x200_FW_SERVICE_PUMP2_STOPCMD : fbDO_IF;  (* Signal conditioning module *)
    x200_FW_STORAGE_TANK_DRAINVALVE_CLOSECMD : fbDO_IF;  (* Signal conditioning module *)
    x200_FW_STORAGE_TANK_DRAINVALVE_OPENCMD : fbDO_IF;  (* Signal conditioning module *)
    x200_FW_STORAGE_TANK_FILLVALVE_CLOSECMD : fbDO_IF;  (* Signal conditioning module *)
    x200_FW_STORAGE_TANK_FILLVALVE_OPENCMD : fbDO_IF;  (* Signal conditioning module *)
    x200_FW_SERVICE_TANK_DRAINVALVE_CLOSECMD : fbDO_IF;  (* Signal conditioning module *)
    x200_FW_SERVICE_TANK_DRAINVALVE_OPENCMD : fbDO_IF;  (* Signal conditioning module *)
    x200_FW_SERVICE_TANK_FILLVALVE_CLOSECMD : fbDO_IF;  (* Signal conditioning module *)
    x200_FW_SERVICE_TANK_FILLVALVE_OPENCMD : fbDO_IF;  (* Signal conditioning module *)
    x100_IGNITOR_ACTIVATE_CMD : fbDO_IF;  (* Signal conditioning module *)
    x100_BLOWER_MOTOR_START_CMD : fbDO_IF;  (* Signal conditioning module *)
    x100_MAIN_FUEL_VALVE_CLOSE_CMD : fbDO_IF;  (* Signal conditioning module *)
    x100_MAIN_FUEL_VALVE_OPEN_CMD : fbDO_IF;  (* Signal conditioning module *)
    x300_HFO_HEATING_VALVE_CLOSE_CMD : fbDO_IF;  (* Signal conditioning module *)
    x300_HFO_HEATING_VALVE_OPEN_CMD : fbDO_IF;  (* Signal conditioning module *)
    x300_HVAC_HEATING_VALVE_CLOSE_CMD : fbDO_IF;  (* Signal conditioning module *)
    x300_HVAC_HEATING_VALVE_OPEN_CMD : fbDO_IF;  (* Signal conditioning module *)
    x300_OPERATIONAL_CONSUMERS_VALVE_CLOSE_CMD : fbDO_IF;  (* Signal conditioning module *)
    x300_OPERATIONAL_CONSUMERS_VALVE_OPEN_CMD : fbDO_IF;  (* Signal conditioning module *)
  END_VAR

                    IF NOT GVL.SIMULATE THEN
x200_FW_SERVICE_PUMP1_STARTCMD(SignalConn := IO.DOS.x200_FW_SERVICE_PUMP1_STARTCMD);
x200_FW_SERVICE_PUMP1_STOPCMD(SignalConn := IO.DOS.x200_FW_SERVICE_PUMP1_STOPCMD);
x200_FW_SERVICE_PUMP2_STARTCMD(SignalConn := IO.DOS.x200_FW_SERVICE_PUMP2_STARTCMD);
x200_FW_SERVICE_PUMP2_STOPCMD(SignalConn := IO.DOS.x200_FW_SERVICE_PUMP2_STOPCMD);
x200_FW_STORAGE_TANK_DRAINVALVE_CLOSECMD(SignalConn := IO.DOS.x200_FW_STORAGE_TANK_DRAINVALVE_CLOSECMD);
x200_FW_STORAGE_TANK_DRAINVALVE_OPENCMD(SignalConn := IO.DOS.x200_FW_STORAGE_TANK_DRAINVALVE_OPENCMD);
x200_FW_STORAGE_TANK_FILLVALVE_CLOSECMD(SignalConn := IO.DOS.x200_FW_STORAGE_TANK_FILLVALVE_CLOSECMD);
x200_FW_STORAGE_TANK_FILLVALVE_OPENCMD(SignalConn := IO.DOS.x200_FW_STORAGE_TANK_FILLVALVE_OPENCMD);
x200_FW_SERVICE_TANK_DRAINVALVE_CLOSECMD(SignalConn := IO.DOS.x200_FW_SERVICE_TANK_DRAINVALVE_CLOSECMD);
x200_FW_SERVICE_TANK_DRAINVALVE_OPENCMD(SignalConn := IO.DOS.x200_FW_SERVICE_TANK_DRAINVALVE_OPENCMD);
x200_FW_SERVICE_TANK_FILLVALVE_CLOSECMD(SignalConn := IO.DOS.x200_FW_SERVICE_TANK_FILLVALVE_CLOSECMD);
x200_FW_SERVICE_TANK_FILLVALVE_OPENCMD(SignalConn := IO.DOS.x200_FW_SERVICE_TANK_FILLVALVE_OPENCMD);
x100_IGNITOR_ACTIVATE_CMD(SignalConn := IO.DOS.x100_IGNITOR_ACTIVATE_CMD);
x100_BLOWER_MOTOR_START_CMD(SignalConn := IO.DOS.x100_BLOWER_MOTOR_START_CMD);
x100_MAIN_FUEL_VALVE_CLOSE_CMD(SignalConn := IO.DOS.x100_MAIN_FUEL_VALVE_CLOSE_CMD);
x100_MAIN_FUEL_VALVE_OPEN_CMD(SignalConn := IO.DOS.x100_MAIN_FUEL_VALVE_OPEN_CMD);
x300_HFO_HEATING_VALVE_CLOSE_CMD(SignalConn := IO.DOS.x300_HFO_HEATING_VALVE_CLOSE_CMD);
x300_HFO_HEATING_VALVE_OPEN_CMD(SignalConn := IO.DOS.x300_HFO_HEATING_VALVE_OPEN_CMD);
x300_HVAC_HEATING_VALVE_CLOSE_CMD(SignalConn := IO.DOS.x300_HVAC_HEATING_VALVE_CLOSE_CMD);
x300_HVAC_HEATING_VALVE_OPEN_CMD(SignalConn := IO.DOS.x300_HVAC_HEATING_VALVE_OPEN_CMD);
x300_OPERATIONAL_CONSUMERS_VALVE_CLOSE_CMD(SignalConn := IO.DOS.x300_OPERATIONAL_CONSUMERS_VALVE_CLOSE_CMD);
x300_OPERATIONAL_CONSUMERS_VALVE_OPEN_CMD(SignalConn := IO.DOS.x300_OPERATIONAL_CONSUMERS_VALVE_OPEN_CMD);

END_IF
                  
END_PROGRAM

PROGRAM DIS_POU
  VAR
    x100_PHOTOCELL1_ACTIVE : fbDI_IF;  (* Signal conditioning module *)
    x100_PHOTOCELL2_ACTIVE : fbDI_IF;  (* Signal conditioning module *)
    x100_BURNER_DOOR_OPEN : fbDI_IF;  (* Signal conditioning module *)
    x100_IGNITION_COIL_ACTIVATED : fbDI_IF;  (* Signal conditioning module *)
    x100_MAIN_FUEL_VALVE_CLOSED : fbDI_IF;  (* Signal conditioning module *)
    x100_MAIN_FUEL_VALVE_OPEN : fbDI_IF;  (* Signal conditioning module *)
    x200_FW_STORAGE_TK_HLIMITSWITCH : fbDI_IF;  (* Signal conditioning module *)
    x200_FW_STORAGE_TK_LLIMITSWITCH : fbDI_IF;  (* Signal conditioning module *)
    x200_FW_SERVICE_PUMP2_RUNNING : fbDI_IF;  (* Signal conditioning module *)
    x200_FW_SERVICE_PUMP2_STOPPED : fbDI_IF;  (* Signal conditioning module *)
    x200_FW_SERVICE_PUMP2_READY : fbDI_IF;  (* Signal conditioning module *)
    x200_FW_SERVICE_PUMP2_TRIPPED : fbDI_IF;  (* Signal conditioning module *)
    x200_FW_SERVICE_PUMP2_REMOTE : fbDI_IF;  (* Signal conditioning module *)
    x200_FW_SERVICE_PUMP1_RUNNING : fbDI_IF;  (* Signal conditioning module *)
    x200_FW_SERVICE_PUMP1_STOPPED : fbDI_IF;  (* Signal conditioning module *)
    x200_FW_SERVICE_PUMP1_READY : fbDI_IF;  (* Signal conditioning module *)
    x200_FW_SERVICE_PUMP1_TRIPPED : fbDI_IF;  (* Signal conditioning module *)
    x200_FW_SERVICE_PUMP1_REMOTE : fbDI_IF;  (* Signal conditioning module *)
    x200_FW_STORAGE_TK_DRAINVALVE_CLOSED : fbDI_IF;  (* Signal conditioning module *)
    x200_FW_STORAGE_TK_DRAINVALVE_OPENED : fbDI_IF;  (* Signal conditioning module *)
    x200_FW_STORAGE_TK_DRAINVALVE_READY : fbDI_IF;  (* Signal conditioning module *)
    x200_FW_STORAGE_TK_DRAINVALVE_REMOTE : fbDI_IF;  (* Signal conditioning module *)
    x200_FW_STORAGE_TK_FILLVALVE_CLOSED : fbDI_IF;  (* Signal conditioning module *)
    x200_FW_STORAGE_TK_FILLVALVE_OPENED : fbDI_IF;  (* Signal conditioning module *)
    x200_FW_STORAGE_TK_FILLVALVE_READY : fbDI_IF;  (* Signal conditioning module *)
    x200_FW_STORAGE_TK_FILLVALVE_REMOTE : fbDI_IF;  (* Signal conditioning module *)
    x200_FW_SERVICE_TK_HLIMITSWITCH : fbDI_IF;  (* Signal conditioning module *)
    x200_FW_SERVICE_TK_LLIMITSWITCH : fbDI_IF;  (* Signal conditioning module *)
    x200_FW_SERVICE_TK_DRAINVALVE_CLOSED : fbDI_IF;  (* Signal conditioning module *)
    x200_FW_SERVICE_TK_DRAINVALVE_OPENED : fbDI_IF;  (* Signal conditioning module *)
    x200_FW_SERVICE_TK_DRAINVALVE_READY : fbDI_IF;  (* Signal conditioning module *)
    x200_FW_SERVICE_TK_DRAINVALVE_REMOTE : fbDI_IF;  (* Signal conditioning module *)
    x200_FW_SERVICE_TK_FILLVALVE_CLOSED : fbDI_IF;  (* Signal conditioning module *)
    x200_FW_SERVICE_TK_FILLVALVE_OPENED : fbDI_IF;  (* Signal conditioning module *)
    x200_FW_SERVICE_TK_FILLVALVE_READY : fbDI_IF;  (* Signal conditioning module *)
    x200_FW_SERVICE_TK_FILLVALVE_REMOTE : fbDI_IF;  (* Signal conditioning module *)
    x300_OPERATIONAL_CONSUMERS_VALVE_OPEN : fbDI_IF;  (* Signal conditioning module *)
    x300_HFO_HEATING_VALVE_CLOSED : fbDI_IF;  (* Signal conditioning module *)
    x300_HFO_HEATING_VALVE_OPEN : fbDI_IF;  (* Signal conditioning module *)
    x300_HVAC_HEATING_VALVE_CLOSED : fbDI_IF;  (* Signal conditioning module *)
    x300_HVAC_HEATING_VALVE_OPEN : fbDI_IF;  (* Signal conditioning module *)
    x300_OPERATIONAL_CONSUMERS_VALVE_CLOSED : fbDI_IF;  (* Signal conditioning module *)
    x900_EMERGENCY_STOP : fbDI_IF;  (* Signal conditioning module *)
    x900_SYSTEM_REMOTE_SWITCH : fbDI_IF;  (* Signal conditioning module *)
  END_VAR

                    
IF NOT GVL.SIMULATE THEN
x100_PHOTOCELL1_ACTIVE(SignalConn => IO.DIS.x100_PHOTOCELL1_ACTIVE);
x100_PHOTOCELL2_ACTIVE(SignalConn => IO.DIS.x100_PHOTOCELL2_ACTIVE);
x100_BURNER_DOOR_OPEN(SignalConn => IO.DIS.x100_BURNER_DOOR_OPEN);
x100_IGNITION_COIL_ACTIVATED(SignalConn => IO.DIS.x100_IGNITION_COIL_ACTIVATED);
x100_MAIN_FUEL_VALVE_CLOSED(SignalConn => IO.DIS.x100_MAIN_FUEL_VALVE_CLOSED);
x100_MAIN_FUEL_VALVE_OPEN(SignalConn => IO.DIS.x100_MAIN_FUEL_VALVE_OPEN);
x200_FW_STORAGE_TK_HLIMITSWITCH(SignalConn => IO.DIS.x200_FW_STORAGE_TK_HLIMITSWITCH);
x200_FW_STORAGE_TK_LLIMITSWITCH(SignalConn => IO.DIS.x200_FW_STORAGE_TK_LLIMITSWITCH);
x200_FW_SERVICE_PUMP2_RUNNING(SignalConn => IO.DIS.x200_FW_SERVICE_PUMP2_RUNNING);
x200_FW_SERVICE_PUMP2_STOPPED(SignalConn => IO.DIS.x200_FW_SERVICE_PUMP2_STOPPED);
x200_FW_SERVICE_PUMP2_READY(SignalConn => IO.DIS.x200_FW_SERVICE_PUMP2_READY);
x200_FW_SERVICE_PUMP2_TRIPPED(SignalConn => IO.DIS.x200_FW_SERVICE_PUMP2_TRIPPED);
x200_FW_SERVICE_PUMP2_REMOTE(SignalConn => IO.DIS.x200_FW_SERVICE_PUMP2_REMOTE);
x200_FW_SERVICE_PUMP1_RUNNING(SignalConn => IO.DIS.x200_FW_SERVICE_PUMP1_RUNNING);
x200_FW_SERVICE_PUMP1_STOPPED(SignalConn => IO.DIS.x200_FW_SERVICE_PUMP1_STOPPED);
x200_FW_SERVICE_PUMP1_READY(SignalConn => IO.DIS.x200_FW_SERVICE_PUMP1_READY);
x200_FW_SERVICE_PUMP1_TRIPPED(SignalConn => IO.DIS.x200_FW_SERVICE_PUMP1_TRIPPED);
x200_FW_SERVICE_PUMP1_REMOTE(SignalConn => IO.DIS.x200_FW_SERVICE_PUMP1_REMOTE);
x200_FW_STORAGE_TK_DRAINVALVE_CLOSED(SignalConn => IO.DIS.x200_FW_STORAGE_TK_DRAINVALVE_CLOSED);
x200_FW_STORAGE_TK_DRAINVALVE_OPENED(SignalConn => IO.DIS.x200_FW_STORAGE_TK_DRAINVALVE_OPENED);
x200_FW_STORAGE_TK_DRAINVALVE_READY(SignalConn => IO.DIS.x200_FW_STORAGE_TK_DRAINVALVE_READY);
x200_FW_STORAGE_TK_DRAINVALVE_REMOTE(SignalConn => IO.DIS.x200_FW_STORAGE_TK_DRAINVALVE_REMOTE);
x200_FW_STORAGE_TK_FILLVALVE_CLOSED(SignalConn => IO.DIS.x200_FW_STORAGE_TK_FILLVALVE_CLOSED);
x200_FW_STORAGE_TK_FILLVALVE_OPENED(SignalConn => IO.DIS.x200_FW_STORAGE_TK_FILLVALVE_OPENED);
x200_FW_STORAGE_TK_FILLVALVE_READY(SignalConn => IO.DIS.x200_FW_STORAGE_TK_FILLVALVE_READY);
x200_FW_STORAGE_TK_FILLVALVE_REMOTE(SignalConn => IO.DIS.x200_FW_STORAGE_TK_FILLVALVE_REMOTE);
x200_FW_SERVICE_TK_HLIMITSWITCH(SignalConn => IO.DIS.x200_FW_SERVICE_TK_HLIMITSWITCH);
x200_FW_SERVICE_TK_LLIMITSWITCH(SignalConn => IO.DIS.x200_FW_SERVICE_TK_LLIMITSWITCH);
x200_FW_SERVICE_TK_DRAINVALVE_CLOSED(SignalConn => IO.DIS.x200_FW_SERVICE_TK_DRAINVALVE_CLOSED);
x200_FW_SERVICE_TK_DRAINVALVE_OPENED(SignalConn => IO.DIS.x200_FW_SERVICE_TK_DRAINVALVE_OPENED);
x200_FW_SERVICE_TK_DRAINVALVE_READY(SignalConn => IO.DIS.x200_FW_SERVICE_TK_DRAINVALVE_READY);
x200_FW_SERVICE_TK_DRAINVALVE_REMOTE(SignalConn => IO.DIS.x200_FW_SERVICE_TK_DRAINVALVE_REMOTE);
x200_FW_SERVICE_TK_FILLVALVE_CLOSED(SignalConn => IO.DIS.x200_FW_SERVICE_TK_FILLVALVE_CLOSED);
x200_FW_SERVICE_TK_FILLVALVE_OPENED(SignalConn => IO.DIS.x200_FW_SERVICE_TK_FILLVALVE_OPENED);
x200_FW_SERVICE_TK_FILLVALVE_READY(SignalConn => IO.DIS.x200_FW_SERVICE_TK_FILLVALVE_READY);
x200_FW_SERVICE_TK_FILLVALVE_REMOTE(SignalConn => IO.DIS.x200_FW_SERVICE_TK_FILLVALVE_REMOTE);
x300_OPERATIONAL_CONSUMERS_VALVE_OPEN(SignalConn => IO.DIS.x300_OPERATIONAL_CONSUMERS_VALVE_OPEN);
x300_HFO_HEATING_VALVE_CLOSED(SignalConn => IO.DIS.x300_HFO_HEATING_VALVE_CLOSED);
x300_HFO_HEATING_VALVE_OPEN(SignalConn => IO.DIS.x300_HFO_HEATING_VALVE_OPEN);
x300_HVAC_HEATING_VALVE_CLOSED(SignalConn => IO.DIS.x300_HVAC_HEATING_VALVE_CLOSED);
x300_HVAC_HEATING_VALVE_OPEN(SignalConn => IO.DIS.x300_HVAC_HEATING_VALVE_OPEN);
x300_OPERATIONAL_CONSUMERS_VALVE_CLOSED(SignalConn => IO.DIS.x300_OPERATIONAL_CONSUMERS_VALVE_CLOSED);
x900_EMERGENCY_STOP(SignalConn => IO.DIS.x900_EMERGENCY_STOP);
x900_SYSTEM_REMOTE_SWITCH(SignalConn => IO.DIS.x900_SYSTEM_REMOTE_SWITCH);


END_IF
                  
END_PROGRAM

PROGRAM AIS_POU
  VAR
    x150_BOILER_WATER_LEVEL : fbAI_IF := (CFG := (sigMin := 0, sigMax := 100, Scale := 1));  (* Signal conditioning module *)
    x200_FRESH_WATER_STORAGE_TANK_LEVEL : fbAI_IF := (CFG := (sigMin := 0, sigMax := 100, Scale := 1));  (* Signal conditioning module *)
    x200_FRESH_WATER_SERVICE_TANK_LEVEL : fbAI_IF := (CFG := (sigMin := 0, sigMax := 100, Scale := 1));  (* Signal conditioning module *)
    x300_HFO_HEATING_SYSTEM_CONSUMPTION : fbAI_IF := (CFG := (sigMin := 0, sigMax := 100, Scale := 1));  (* Signal conditioning module *)
    x300_HVAC_SYSTEM_CONSUMPTION : fbAI_IF := (CFG := (sigMin := 0, sigMax := 100, Scale := 1));  (* Signal conditioning module *)
    x300_OPERATIONAL_CONSUMERS_CONSUMPTION : fbAI_IF := (CFG := (sigMin := 0, sigMax := 100, Scale := 1));  (* Signal conditioning module *)
    x300_SYSTEM_STEAM_PRESSURE : fbAI_IF := (CFG := (sigMin := 0, sigMax := 100, Scale := 1));  (* Signal conditioning module *)
  END_VAR

                    IF NOT GVL.SIMULATE THEN
	(*Analog input signal conditioning function block calls *)
	x150_BOILER_WATER_LEVEL(SignalConn => IO.AIS.x150_BOILER_WATER_LEVEL);
	x200_FRESH_WATER_STORAGE_TANK_LEVEL(SignalConn => IO.AIS.x200_FRESH_WATER_STORAGE_TANK_LEVEL);
	x200_FRESH_WATER_SERVICE_TANK_LEVEL(SignalConn => IO.AIS.x200_FRESH_WATER_SERVICE_TANK_LEVEL);
	x300_HFO_HEATING_SYSTEM_CONSUMPTION(SignalConn => IO.AIS.x300_HFO_HEATING_SYSTEM_CONSUMPTION);
	x300_HVAC_SYSTEM_CONSUMPTION(SignalConn => IO.AIS.x300_HVAC_SYSTEM_CONSUMPTION);
	x300_OPERATIONAL_CONSUMERS_CONSUMPTION(SignalConn => IO.AIS.x300_OPERATIONAL_CONSUMERS_CONSUMPTION);
	x300_SYSTEM_STEAM_PRESSURE(SignalConn => IO.AIS.x300_SYSTEM_STEAM_PRESSURE);
END_IF
                  
END_PROGRAM

CONFIGURATION Device
  RESOURCE Application ON PLC
    {attribute 'qualified_only'}
    VAR_GLOBAL  (* IO *)
      AIS : AIS_Typ;  (* Analog input structure *)
      AOS : AOS_Typ;  (* Analog output structure *)
      DIS : DIS_Typ;  (* Digital input structure *)
      DOS : DOS_Typ;  (* Digital output structure *)
    END_VAR
    {attribute 'qualified_only'}
    VAR_GLOBAL  (* GVL *)
      SIMULATE : BOOL := TRUE;  (* Turns on simulation mode in the software *)
    END_VAR
    TASK MainTask(INTERVAL := T#20ms, PRIORITY := 1);
    TASK VISU_TASK(INTERVAL := T#100ms, PRIORITY := 31);
    TASK TrendRecordingTask(INTERVAL := T#100ms, PRIORITY := 31);
    PROGRAM AOS_POU WITH MainTask : AOS_POU;
    PROGRAM DIS_POU WITH MainTask : DIS_POU;
    PROGRAM DOS_POU WITH MainTask : DOS_POU;
    PROGRAM AIS_POU WITH MainTask : AIS_POU;
    PROGRAM Main WITH MainTask : Main;
    PROGRAM Simulator WITH MainTask : Simulator;
    PROGRAM VisuElems.Visu_Prg WITH VISU_TASK : VisuElems.Visu_Prg;
  END_RESOURCE
END_CONFIGURATION
